LIN {X 0,Y 192.943,Z 262.908,A -85,B 0,C 180,E1 -21964.191,E2 -21964.191} C_VEL
LIN {X 0,Y 193.037,Z 262.919,A -85,B 0,C 180,E1 -21968.387,E2 -21968.387} C_VEL
LIN {X 0,Y 192.808,Z 262.969,A -85,B 0,C 180,E1 -21972.646,E2 -21972.646} C_VEL
LIN {X 0,Y 192.733,Z 262.955,A -85,B 0,C 180,E1 -21976.974,E2 -21976.974} C_VEL
LIN {X 0,Y 192.605,Z 262.981,A -85,B 0,C 180,E1 -21981.414,E2 -21981.414} C_VEL
LIN {X 0,Y 192.66,Z 262.986,A -85,B 0,C 180,E1 -21984.214,E2 -21984.214} C_VEL
LIN {X 0,Y 192.628,Z 262.969,A -85,B 0,C 180,E1 -21988.874,E2 -21988.874} C_VEL
LIN {X 0,Y 192.623,Z 262.992,A -85,B 0,C 180,E1 -21993.195,E2 -21993.195} C_VEL
LIN {X 0,Y 192.571,Z 262.995,A -85,B 0,C 180,E1 -21998.362,E2 -21998.362} C_VEL
LIN {X 0,Y 192.501,Z 262.997,A -85,B 0,C 180,E1 -22003.094,E2 -22003.094} C_VEL
LIN {X 0,Y 192.501,Z 262.997,A -85,B 0,C 180,E1 -22006.917,E2 -22006.917} C_VEL
LIN {X 0,Y 192.636,Z 263.112,A -85,B 0,C 180,E1 -22011.215,E2 -22011.215} C_VEL
LIN {X 0,Y 193.486,Z 266.81,A -85,B 0,C 180,E1 -22013.229,E2 -22013.229} C_VEL
LIN {X 0,Y 195.559,Z 272.184,A -85,B 0,C 180,E1 -22013.906,E2 -22013.906} C_VEL
LIN {X 0,Y 202.679,Z 290.586,A -85,B 0,C 180,E1 -22015.768,E2 -22015.768} C_VEL
LIN {X 0,Y 207.241,Z 304.045,A -85,B 0,C 180,E1 -22016.961,E2 -22016.961} C_VEL
LIN {X 0,Y 208.938,Z 318.725,A -85,B 0,C 180,E1 -22017.817,E2 -22017.817} C_VEL
LIN {X 0,Y 208.478,Z 329.306,A -85,B 0,C 180,E1 -22018.229,E2 -22018.229} C_VEL
LIN {X 0,Y 207.471,Z 335.115,A -85,B 0,C 180,E1 -22018.369,E2 -22018.369} C_VEL
LIN {X 0,Y 201.296,Z 353.95,A -85,B 0,C 180,E1 -22018.502,E2 -22018.502} C_VEL
LIN {X 0,Y 200.376,Z 359.758,A -85,B 0,C 180,E1 -22018.662,E2 -22018.662} C_VEL
LIN {X 0,Y 199.212,Z 377.564,A -85,B 0,C 180,E1 -22019.45,E2 -22019.45} C_VEL
LIN {X 0,Y 198.023,Z 389.93,A -85,B 0,C 180,E1 -22020.35,E2 -22020.35} C_VEL
LIN {X 0,Y 196.332,Z 402.666,A -85,B 0,C 180,E1 -22021.682,E2 -22021.682} C_VEL
LIN {X 0,Y 194.124,Z 414.844,A -85,B 0,C 180,E1 -22023.38,E2 -22023.38} C_VEL
LIN {X 0,Y 192.053,Z 425.896,A -85,B 0,C 180,E1 -22025.398,E2 -22025.398} C_VEL
LIN {X 0,Y 189.821,Z 436.544,A -85,B 0,C 180,E1 -22027.884,E2 -22027.884} C_VEL
LIN {X 0,Y 188.046,Z 444.993,A -85,B 0,C 180,E1 -22030.341,E2 -22030.341} C_VEL
LIN {X 0,Y 186.127,Z 453.853,A -85,B 0,C 180,E1 -22033.545,E2 -22033.545} C_VEL
LIN {X 0,Y 184.71,Z 460.891,A -85,B 0,C 180,E1 -22036.8,E2 -22036.8} C_VEL
LIN {X 0,Y 183.77,Z 466.502,A -85,B 0,C 180,E1 -22040.087,E2 -22040.087} C_VEL
LIN {X 0,Y 183.246,Z 470.863,A -85,B 0,C 180,E1 -22043.389,E2 -22043.389} C_VEL
LIN {X 0,Y 183.046,Z 474.187,A -85,B 0,C 180,E1 -22046.805,E2 -22046.805} C_VEL
LIN {X 0,Y 183.098,Z 476.306,A -85,B 0,C 180,E1 -22049.996,E2 -22049.996} C_VEL
LIN {X 0,Y 182.998,Z 477.475,A -85,B 0,C 180,E1 -22052.916,E2 -22052.916} C_VEL
LIN {X 0,Y 183.265,Z 477.907,A -85,B 0,C 180,E1 -22056.602,E2 -22056.602} C_VEL
LIN {X 0,Y 184.266,Z 476.962,A -85,B 0,C 180,E1 -22060.99,E2 -22060.99} C_VEL
LIN {X 0,Y 186.161,Z 474.469,A -85,B 0,C 180,E1 -22065.319,E2 -22065.319} C_VEL
LIN {X 0,Y 188.203,Z 471.507,A -85,B 0,C 180,E1 -22068.502,E2 -22068.502} C_VEL
LIN {X 0,Y 191.01,Z 467.529,A -85,B 0,C 180,E1 -22071.584,E2 -22071.584} C_VEL
LIN {X 0,Y 194.38,Z 462.447,A -85,B 0,C 180,E1 -22074.565,E2 -22074.565} C_VEL
LIN {X 0,Y 197.93,Z 456.142,A -85,B 0,C 180,E1 -22077.486,E2 -22077.486} C_VEL
LIN {X 0,Y 202.122,Z 448.306,A -85,B 0,C 180,E1 -22080.273,E2 -22080.273} C_VEL
LIN {X 0,Y 206.964,Z 438.674,A -85,B 0,C 180,E1 -22082.906,E2 -22082.906} C_VEL
LIN {X 0,Y 211.367,Z 428.74,A -85,B 0,C 180,E1 -22084.995,E2 -22084.995} C_VEL
LIN {X 0,Y 215.507,Z 417.692,A -85,B 0,C 180,E1 -22086.811,E2 -22086.811} C_VEL
LIN {X 0,Y 219.025,Z 406.97,A -85,B 0,C 180,E1 -22088.143,E2 -22088.143} C_VEL
LIN {X 0,Y 222.085,Z 395.375,A -85,B 0,C 180,E1 -22089.26,E2 -22089.26} C_VEL
LIN {X 0,Y 224.719,Z 382.374,A -85,B 0,C 180,E1 -22090.145,E2 -22090.145} C_VEL
LIN {X 0,Y 226.623,Z 368.194,A -85,B 0,C 180,E1 -22090.777,E2 -22090.777} C_VEL
LIN {X 0,Y 229.852,Z 331.704,A -85,B 0,C 180,E1 -22092.063,E2 -22092.063} C_VEL
LIN {X 0,Y 226.618,Z 323.344,A -85,B 0,C 180,E1 -22093.846,E2 -22093.846} C_VEL
LIN {X 0,Y 222.913,Z 315.251,A -85,B 0,C 180,E1 -22096.011,E2 -22096.011} C_VEL
LIN {X 0,Y 219.308,Z 308.517,A -85,B 0,C 180,E1 -22098.305,E2 -22098.305} C_VEL
LIN {X 0,Y 217.579,Z 305.452,A -85,B 0,C 180,E1 -22099.541,E2 -22099.541} C_VEL
LIN {X 0,Y 215.143,Z 301.303,A -85,B 0,C 180,E1 -22101.43,E2 -22101.43} C_VEL
LIN {X 0,Y 212.377,Z 296.664,A -85,B 0,C 180,E1 -22103.944,E2 -22103.944} C_VEL
LIN {X 0,Y 208.556,Z 290.768,A -85,B 0,C 180,E1 -22108.479,E2 -22108.479} C_VEL
LIN {X 0,Y 205.607,Z 286.729,A -85,B 0,C 180,E1 -22115.057,E2 -22115.057} C_VEL
LIN {X 0,Y 205.277,Z 286.197,A -85,B 0,C 180,E1 -22117.864,E2 -22117.864} C_VEL
LIN {X 0,Y 206.045,Z 286.988,A -85,B 0,C 180,E1 -22122.742,E2 -22122.742} C_VEL
LIN {X 0,Y 209.265,Z 290.496,A -85,B 0,C 180,E1 -22128.554,E2 -22128.554} C_VEL
LIN {X 0,Y 212.901,Z 295.629,A -85,B 0,C 180,E1 -22132.601,E2 -22132.601} C_VEL
LIN {X 0,Y 215.785,Z 299.597,A -85,B 0,C 180,E1 -22135.063,E2 -22135.063} C_VEL
LIN {X 0,Y 218.709,Z 304.458,A -85,B 0,C 180,E1 -22137.267,E2 -22137.267} C_VEL
LIN {X 0,Y 223.96,Z 314.057,A -85,B 0,C 180,E1 -22140.63,E2 -22140.63} C_VEL
LIN {X 0,Y 227.578,Z 321.869,A -85,B 0,C 180,E1 -22142.69,E2 -22142.69} C_VEL
LIN {X 0,Y 230.089,Z 328.091,A -85,B 0,C 180,E1 -22144.05,E2 -22144.05} C_VEL
LIN {X 0,Y 226.135,Z 370.908,A -85,B 0,C 180,E1 -22145.586,E2 -22145.586} C_VEL
LIN {X 0,Y 224.019,Z 383.993,A -85,B 0,C 180,E1 -22146.304,E2 -22146.304} C_VEL
LIN {X 0,Y 221.324,Z 396.216,A -85,B 0,C 180,E1 -22147.285,E2 -22147.285} C_VEL
LIN {X 0,Y 217.858,Z 408.634,A -85,B 0,C 180,E1 -22148.685,E2 -22148.685} C_VEL
LIN {X 0,Y 213.843,Z 420.129,A -85,B 0,C 180,E1 -22150.369,E2 -22150.369} C_VEL
LIN {X 0,Y 210.115,Z 429.29,A -85,B 0,C 180,E1 -22152.088,E2 -22152.088} C_VEL
LIN {X 0,Y 206.133,Z 437.969,A -85,B 0,C 180,E1 -22154.132,E2 -22154.132} C_VEL
LIN {X 0,Y 201.879,Z 446.182,A -85,B 0,C 180,E1 -22156.578,E2 -22156.578} C_VEL
LIN {X 0,Y 197.216,Z 454.354,A -85,B 0,C 180,E1 -22159.727,E2 -22159.727} C_VEL
LIN {X 0,Y 193.229,Z 460.737,A -85,B 0,C 180,E1 -22163,E2 -22163} C_VEL
LIN {X 0,Y 189.936,Z 465.541,A -85,B 0,C 180,E1 -22166.343,E2 -22166.343} C_VEL
LIN {X 0,Y 187.035,Z 469.436,A -85,B 0,C 180,E1 -22170.212,E2 -22170.212} C_VEL
LIN {X 0,Y 185.258,Z 471.55,A -85,B 0,C 180,E1 -22173.434,E2 -22173.434} C_VEL
LIN {X 0,Y 183.606,Z 472.976,A -85,B 0,C 180,E1 -22177.745,E2 -22177.745} C_VEL
LIN {X 0,Y 183,Z 473.017,A -85,B 0,C 180,E1 -22180.736,E2 -22180.736} C_VEL
LIN {X 0,Y 182.634,Z 472.317,A -85,B 0,C 180,E1 -22183.817,E2 -22183.817} C_VEL
LIN {X 0,Y 182.538,Z 470.782,A -85,B 0,C 180,E1 -22186.989,E2 -22186.989} C_VEL
LIN {X 0,Y 182.746,Z 468.284,A -85,B 0,C 180,E1 -22190.251,E2 -22190.251} C_VEL
LIN {X 0,Y 183.32,Z 464.679,A -85,B 0,C 180,E1 -22193.589,E2 -22193.589} C_VEL
LIN {X 0,Y 184.166,Z 459.647,A -85,B 0,C 180,E1 -22197.059,E2 -22197.059} C_VEL
LIN {X 0,Y 185.489,Z 452.98,A -85,B 0,C 180,E1 -22200.591,E2 -22200.591} C_VEL
LIN {X 0,Y 187.055,Z 445.451,A -85,B 0,C 180,E1 -22203.738,E2 -22203.738} C_VEL
LIN {X 0,Y 188.731,Z 437.834,A -85,B 0,C 180,E1 -22206.304,E2 -22206.304} C_VEL
LIN {X 0,Y 190.794,Z 428.078,A -85,B 0,C 180,E1 -22208.956,E2 -22208.956} C_VEL
LIN {X 0,Y 192.965,Z 417.676,A -85,B 0,C 180,E1 -22211.199,E2 -22211.199} C_VEL
LIN {X 0,Y 194.794,Z 407.505,A -85,B 0,C 180,E1 -22212.958,E2 -22212.958} C_VEL
LIN {X 0,Y 196.748,Z 395.175,A -85,B 0,C 180,E1 -22214.614,E2 -22214.614} C_VEL
LIN {X 0,Y 198.396,Z 381.535,A -85,B 0,C 180,E1 -22215.941,E2 -22215.941} C_VEL
LIN {X 0,Y 199.661,Z 367.958,A -85,B 0,C 180,E1 -22216.81,E2 -22216.81} C_VEL
LIN {X 0,Y 202.729,Z 307.987,A -85,B 0,C 180,E1 -22219.215,E2 -22219.215} C_VEL
LIN {X 0,Y 195.715,Z 287.677,A -85,B 0,C 180,E1 -22221.114,E2 -22221.114} C_VEL
LIN {X 0,Y 189.308,Z 271.417,A -85,B 0,C 180,E1 -22222.874,E2 -22222.874} C_VEL
LIN {X 0,Y 186.118,Z 264.918,A -85,B 0,C 180,E1 -22223.771,E2 -22223.771} C_VEL
LIN {X 0,Y 185.888,Z 263.91,A -85,B 0,C 180,E1 -22224.24,E2 -22224.24} C_VEL
LIN {X 0,Y 186.167,Z 263.797,A -85,B 0,C 180,E1 -22227.84,E2 -22227.84} C_VEL
LIN {X 0,Y 186.349,Z 263.764,A -85,B 0,C 180,E1 -22230.004,E2 -22230.004} C_VEL
LIN {X 0,Y 185.876,Z 263.818,A -85,B 0,C 180,E1 -22234.341,E2 -22234.341} C_VEL
LIN {X 0,Y 185.949,Z 263.814,A -85,B 0,C 180,E1 -22238.699,E2 -22238.699} C_VEL
LIN {X 0,Y 185.669,Z 263.855,A -85,B 0,C 180,E1 -22243.131,E2 -22243.131} C_VEL
LIN {X 0,Y 185.633,Z 263.839,A -85,B 0,C 180,E1 -22247.634,E2 -22247.634} C_VEL
LIN {X 0,Y 185.526,Z 263.875,A -85,B 0,C 180,E1 -22252.264,E2 -22252.264} C_VEL
LIN {X 0,Y 185.511,Z 263.851,A -85,B 0,C 180,E1 -22257.044,E2 -22257.044} C_VEL
LIN {X 0,Y 185.533,Z 263.838,A -85,B 0,C 180,E1 -22259.505,E2 -22259.505} C_VEL
LIN {X 0,Y 185.479,Z 263.881,A -85,B 0,C 180,E1 -22264.64,E2 -22264.64} C_VEL
LIN {X 0,Y 185.53,Z 263.87,A -85,B 0,C 180,E1 -22267.327,E2 -22267.327} C_VEL
LIN {X 0,Y 185.526,Z 263.872,A -85,B 0,C 180,E1 -22270.771,E2 -22270.771} C_VEL
LIN {X 0,Y 185.554,Z 263.861,A -85,B 0,C 180,E1 -22276.029,E2 -22276.029} C_VEL
LIN {X 0,Y 185.553,Z 263.869,A -85,B 0,C 180,E1 -22279.939,E2 -22279.939} C_VEL
LIN {X 0,Y 185.551,Z 263.868,A -85,B 0,C 180,E1 -22282.719,E2 -22282.719} C_VEL
LIN {X 0,Y 185.521,Z 263.872,A -85,B 0,C 180,E1 -22287.99,E2 -22287.99} C_VEL
LIN {X 0,Y 185.564,Z 263.87,A -85,B 0,C 180,E1 -22290.592,E2 -22290.592} C_VEL
LIN {X 0,Y 185.568,Z 263.856,A -85,B 0,C 180,E1 -22295.397,E2 -22295.397} C_VEL
LIN {X 0,Y 185.618,Z 263.86,A -85,B 0,C 180,E1 -22301.194,E2 -22301.194} C_VEL
LIN {X 0,Y 185.664,Z 263.844,A -85,B 0,C 180,E1 -22304.65,E2 -22304.65} C_VEL
LIN {X 0,Y 185.889,Z 263.83,A -85,B 0,C 180,E1 -22309.435,E2 -22309.435} C_VEL
LIN {X 0,Y 185.936,Z 263.809,A -85,B 0,C 180,E1 -22313.504,E2 -22313.504} C_VEL
LIN {X 0,Y 186.187,Z 263.794,A -85,B 0,C 180,E1 -22317.851,E2 -22317.851} C_VEL
LIN {X 0,Y 186.388,Z 263.76,A -85,B 0,C 180,E1 -22320.014,E2 -22320.014} C_VEL
LIN {X 0,Y 185.892,Z 263.783,A -85,B 0,C 180,E1 -22324.35,E2 -22324.35} C_VEL
LIN {X 0,Y 185.987,Z 263.798,A -85,B 0,C 180,E1 -22328.707,E2 -22328.707} C_VEL
LIN {X 0,Y 185.734,Z 263.848,A -85,B 0,C 180,E1 -22333.136,E2 -22333.136} C_VEL
LIN {X 0,Y 185.672,Z 263.828,A -85,B 0,C 180,E1 -22337.64,E2 -22337.64} C_VEL
LIN {X 0,Y 185.577,Z 263.863,A -85,B 0,C 180,E1 -22342.268,E2 -22342.268} C_VEL
LIN {X 0,Y 185.603,Z 263.867,A -85,B 0,C 180,E1 -22344.656,E2 -22344.656} C_VEL
LIN {X 0,Y 185.571,Z 263.849,A -85,B 0,C 180,E1 -22349.509,E2 -22349.509} C_VEL
LIN {X 0,Y 185.526,Z 263.867,A -85,B 0,C 180,E1 -22354.641,E2 -22354.641} C_VEL
LIN {X 0,Y 185.53,Z 263.86,A -85,B 0,C 180,E1 -22357.322,E2 -22357.322} C_VEL
LIN {X 0,Y 185.487,Z 263.875,A -85,B 0,C 180,E1 -22360.726,E2 -22360.726} C_VEL
LIN {X 0,Y 185.471,Z 263.874,A -85,B 0,C 180,E1 -22366.068,E2 -22366.068} C_VEL
LIN {X 0,Y 185.54,Z 263.987,A -85,B 0,C 180,E1 -22370.564,E2 -22370.564} C_VEL
LIN {X 0,Y 186.251,Z 266.867,A -85,B 0,C 180,E1 -22372.141,E2 -22372.141} C_VEL
LIN {X 0,Y 194.045,Z 286.32,A -85,B 0,C 180,E1 -22374.371,E2 -22374.371} C_VEL
LIN {X 0,Y 200.783,Z 305.431,A -85,B 0,C 180,E1 -22376.209,E2 -22376.209} C_VEL
LIN {X 0,Y 202.406,Z 318.992,A -85,B 0,C 180,E1 -22377.042,E2 -22377.042} C_VEL
LIN {X 0,Y 200.376,Z 359.758,A -85,B 0,C 180,E1 -22378.662,E2 -22378.662} C_VEL
LIN {X 0,Y 199.401,Z 365.56,A -85,B 0,C 180,E1 -22378.812,E2 -22378.812} C_VEL
LIN {X 0,Y 196.096,Z 374.906,A -85,B 0,C 180,E1 -22378.919,E2 -22378.919} C_VEL
LIN {X 0,Y 192.64,Z 384.148,A -85,B 0,C 180,E1 -22379.212,E2 -22379.212} C_VEL
LIN {X 0,Y 191.389,Z 389.784,A -85,B 0,C 180,E1 -22379.607,E2 -22379.607} C_VEL
LIN {X 0,Y 189.738,Z 401.969,A -85,B 0,C 180,E1 -22380.908,E2 -22380.908} C_VEL
LIN {X 0,Y 187.446,Z 414.254,A -85,B 0,C 180,E1 -22382.655,E2 -22382.655} C_VEL
LIN {X 0,Y 185.304,Z 425.407,A -85,B 0,C 180,E1 -22384.739,E2 -22384.739} C_VEL
LIN {X 0,Y 183.36,Z 434.733,A -85,B 0,C 180,E1 -22386.938,E2 -22386.938} C_VEL
LIN {X 0,Y 181.356,Z 443.789,A -85,B 0,C 180,E1 -22389.584,E2 -22389.584} C_VEL
LIN {X 0,Y 179.309,Z 452.844,A -85,B 0,C 180,E1 -22392.901,E2 -22392.901} C_VEL
LIN {X 0,Y 177.746,Z 460.082,A -85,B 0,C 180,E1 -22396.273,E2 -22396.273} C_VEL
LIN {X 0,Y 176.773,Z 465.831,A -85,B 0,C 180,E1 -22399.69,E2 -22399.69} C_VEL
LIN {X 0,Y 176.174,Z 470.315,A -85,B 0,C 180,E1 -22403.123,E2 -22403.123} C_VEL
LIN {X 0,Y 175.945,Z 474.169,A -85,B 0,C 180,E1 -22407.192,E2 -22407.192} C_VEL
LIN {X 0,Y 176.01,Z 476.003,A -85,B 0,C 180,E1 -22409.996,E2 -22409.996} C_VEL
LIN {X 0,Y 175.927,Z 477.13,A -85,B 0,C 180,E1 -22412.685,E2 -22412.685} C_VEL
LIN {X 0,Y 176.197,Z 477.809,A -85,B 0,C 180,E1 -22416.869,E2 -22416.869} C_VEL
LIN {X 0,Y 176.661,Z 477.609,A -85,B 0,C 180,E1 -22419.152,E2 -22419.152} C_VEL
LIN {X 0,Y 178.159,Z 476.029,A -85,B 0,C 180,E1 -22423.687,E2 -22423.687} C_VEL
LIN {X 0,Y 179.295,Z 474.667,A -85,B 0,C 180,E1 -22425.921,E2 -22425.921} C_VEL
LIN {X 0,Y 181.486,Z 471.823,A -85,B 0,C 180,E1 -22429.213,E2 -22429.213} C_VEL
LIN {X 0,Y 184.449,Z 467.979,A -85,B 0,C 180,E1 -22432.393,E2 -22432.393} C_VEL
LIN {X 0,Y 187.984,Z 463.04,A -85,B 0,C 180,E1 -22435.459,E2 -22435.459} C_VEL
LIN {X 0,Y 191.723,Z 456.951,A -85,B 0,C 180,E1 -22438.455,E2 -22438.455} C_VEL
LIN {X 0,Y 196.098,Z 449.433,A -85,B 0,C 180,E1 -22441.305,E2 -22441.305} C_VEL
LIN {X 0,Y 201.13,Z 440.041,A -85,B 0,C 180,E1 -22443.988,E2 -22443.988} C_VEL
LIN {X 0,Y 206.175,Z 429.387,A -85,B 0,C 180,E1 -22446.314,E2 -22446.314} C_VEL
LIN {X 0,Y 210.502,Z 418.502,A -85,B 0,C 180,E1 -22448.14,E2 -22448.14} C_VEL
LIN {X 0,Y 214.636,Z 406.416,A -85,B 0,C 180,E1 -22449.675,E2 -22449.675} C_VEL
LIN {X 0,Y 217.86,Z 394.75,A -85,B 0,C 180,E1 -22450.782,E2 -22450.782} C_VEL
LIN {X 0,Y 220.676,Z 381.375,A -85,B 0,C 180,E1 -22451.664,E2 -22451.664} C_VEL
LIN {X 0,Y 222.481,Z 368.302,A -85,B 0,C 180,E1 -22452.246,E2 -22452.246} C_VEL
LIN {X 0,Y 225.592,Z 334.403,A -85,B 0,C 180,E1 -22453.456,E2 -22453.456} C_VEL
LIN {X 0,Y 222.567,Z 326.486,A -85,B 0,C 180,E1 -22455.273,E2 -22455.273} C_VEL
LIN {X 0,Y 219.169,Z 319.127,A -85,B 0,C 180,E1 -22457.448,E2 -22457.448} C_VEL
LIN {X 0,Y 215.922,Z 312.59,A -85,B 0,C 180,E1 -22459.792,E2 -22459.792} C_VEL
LIN {X 0,Y 213.028,Z 307.584,A -85,B 0,C 180,E1 -22462.111,E2 -22462.111} C_VEL
LIN {X 0,Y 210.548,Z 303.185,A -85,B 0,C 180,E1 -22464.544,E2 -22464.544} C_VEL
LIN {X 0,Y 207.166,Z 297.618,A -85,B 0,C 180,E1 -22468.823,E2 -22468.823} C_VEL
LIN {X 0,Y 204.482,Z 293.758,A -85,B 0,C 180,E1 -22475.153,E2 -22475.153} C_VEL
LIN {X 0,Y 204.165,Z 293.251,A -85,B 0,C 180,E1 -22478.334,E2 -22478.334} C_VEL
LIN {X 0,Y 204.902,Z 293.994,A -85,B 0,C 180,E1 -22482.643,E2 -22482.643} C_VEL
LIN {X 0,Y 207.812,Z 297.302,A -85,B 0,C 180,E1 -22488.157,E2 -22488.157} C_VEL
LIN {X 0,Y 211.121,Z 302.256,A -85,B 0,C 180,E1 -22492.065,E2 -22492.065} C_VEL
LIN {X 0,Y 214.233,Z 306.793,A -85,B 0,C 180,E1 -22494.856,E2 -22494.856} C_VEL
LIN {X 0,Y 216.427,Z 310.764,A -85,B 0,C 180,E1 -22496.588,E2 -22496.588} C_VEL
LIN {X 0,Y 220.877,Z 319.222,A -85,B 0,C 180,E1 -22499.646,E2 -22499.646} C_VEL
LIN {X 0,Y 224.258,Z 326.949,A -85,B 0,C 180,E1 -22501.754,E2 -22501.754} C_VEL
LIN {X 0,Y 225.869,Z 330.944,A -85,B 0,C 180,E1 -22502.676,E2 -22502.676} C_VEL
LIN {X 0,Y 221.927,Z 371.369,A -85,B 0,C 180,E1 -22504.127,E2 -22504.127} C_VEL
LIN {X 0,Y 219.743,Z 384.284,A -85,B 0,C 180,E1 -22504.849,E2 -22504.849} C_VEL
LIN {X 0,Y 216.995,Z 396.09,A -85,B 0,C 180,E1 -22505.796,E2 -22505.796} C_VEL
LIN {X 0,Y 213.768,Z 407.208,A -85,B 0,C 180,E1 -22507.016,E2 -22507.016} C_VEL
LIN {X 0,Y 209.65,Z 418.687,A -85,B 0,C 180,E1 -22508.663,E2 -22508.663} C_VEL
LIN {X 0,Y 205.282,Z 429.112,A -85,B 0,C 180,E1 -22510.589,E2 -22510.589} C_VEL
LIN {X 0,Y 200.874,Z 438.27,A -85,B 0,C 180,E1 -22512.759,E2 -22512.759} C_VEL
LIN {X 0,Y 196.084,Z 446.97,A -85,B 0,C 180,E1 -22515.419,E2 -22515.419} C_VEL
LIN {X 0,Y 191.199,Z 454.924,A -85,B 0,C 180,E1 -22518.602,E2 -22518.602} C_VEL
LIN {X 0,Y 186.853,Z 461.342,A -85,B 0,C 180,E1 -22522.077,E2 -22522.077} C_VEL
LIN {X 0,Y 182.891,Z 466.644,A -85,B 0,C 180,E1 -22526.051,E2 -22526.051} C_VEL
LIN {X 0,Y 180.551,Z 469.49,A -85,B 0,C 180,E1 -22529.096,E2 -22529.096} C_VEL
LIN {X 0,Y 178.038,Z 472.143,A -85,B 0,C 180,E1 -22533.528,E2 -22533.528} C_VEL
LIN {X 0,Y 176.611,Z 473.118,A -85,B 0,C 180,E1 -22537.27,E2 -22537.27} C_VEL
LIN {X 0,Y 175.909,Z 473.08,A -85,B 0,C 180,E1 -22540.622,E2 -22540.622} C_VEL
LIN {X 0,Y 175.524,Z 472.212,A -85,B 0,C 180,E1 -22543.892,E2 -22543.892} C_VEL
LIN {X 0,Y 175.439,Z 470.584,A -85,B 0,C 180,E1 -22547.083,E2 -22547.083} C_VEL
LIN {X 0,Y 175.652,Z 468.211,A -85,B 0,C 180,E1 -22550.201,E2 -22550.201} C_VEL
LIN {X 0,Y 176.163,Z 465.057,A -85,B 0,C 180,E1 -22553.249,E2 -22553.249} C_VEL
LIN {X 0,Y 177.069,Z 459.663,A -85,B 0,C 180,E1 -22557.151,E2 -22557.151} C_VEL
LIN {X 0,Y 178.535,Z 452.539,A -85,B 0,C 180,E1 -22561.043,E2 -22561.043} C_VEL
LIN {X 0,Y 179.934,Z 445.925,A -85,B 0,C 180,E1 -22563.901,E2 -22563.901} C_VEL
LIN {X 0,Y 181.966,Z 437.067,A -85,B 0,C 180,E1 -22566.984,E2 -22566.984} C_VEL
LIN {X 0,Y 184.045,Z 427.574,A -85,B 0,C 180,E1 -22569.612,E2 -22569.612} C_VEL
LIN {X 0,Y 186.201,Z 417.513,A -85,B 0,C 180,E1 -22571.84,E2 -22571.84} C_VEL
LIN {X 0,Y 188.145,Z 407.091,A -85,B 0,C 180,E1 -22573.689,E2 -22573.689} C_VEL
LIN {X 0,Y 190.017,Z 395.658,A -85,B 0,C 180,E1 -22575.273,E2 -22575.273} C_VEL
LIN {X 0,Y 191.719,Z 382.35,A -85,B 0,C 180,E1 -22576.624,E2 -22576.624} C_VEL
LIN {X 0,Y 193.031,Z 368.868,A -85,B 0,C 180,E1 -22577.544,E2 -22577.544} C_VEL
LIN {X 0,Y 196.268,Z 309.645,A -85,B 0,C 180,E1 -22579.989,E2 -22579.989} C_VEL
LIN {X 0,Y 189.484,Z 290.002,A -85,B 0,C 180,E1 -22581.908,E2 -22581.908} C_VEL
LIN {X 0,Y 183.624,Z 274.948,A -85,B 0,C 180,E1 -22583.59,E2 -22583.59} C_VEL
LIN {X 0,Y 179.128,Z 265.97,A -85,B 0,C 180,E1 -22584.868,E2 -22584.868} C_VEL
LIN {X 0,Y 178.868,Z 264.809,A -85,B 0,C 180,E1 -22585.355,E2 -22585.355} C_VEL
LIN {X 0,Y 179.313,Z 264.64,A -85,B 0,C 180,E1 -22590.004,E2 -22590.004} C_VEL
LIN {X 0,Y 178.823,Z 264.696,A -85,B 0,C 180,E1 -22594.512,E2 -22594.512} C_VEL
LIN {X 0,Y 178.879,Z 264.69,A -85,B 0,C 180,E1 -22599.046,E2 -22599.046} C_VEL
LIN {X 0,Y 178.598,Z 264.739,A -85,B 0,C 180,E1 -22603.661,E2 -22603.661} C_VEL
LIN {X 0,Y 178.569,Z 264.719,A -85,B 0,C 180,E1 -22609.222,E2 -22609.222} C_VEL
LIN {X 0,Y 178.472,Z 264.747,A -85,B 0,C 180,E1 -22615.125,E2 -22615.125} C_VEL
LIN {X 0,Y 178.477,Z 264.718,A -85,B 0,C 180,E1 -22620.005,E2 -22620.005} C_VEL
LIN {X 0,Y 178.443,Z 264.757,A -85,B 0,C 180,E1 -22624.231,E2 -22624.231} C_VEL
LIN {X 0,Y 178.436,Z 264.747,A -85,B 0,C 180,E1 -22629.068,E2 -22629.068} C_VEL
LIN {X 0,Y 178.468,Z 264.753,A -85,B 0,C 180,E1 -22632.029,E2 -22632.029} C_VEL
LIN {X 0,Y 178.496,Z 264.743,A -85,B 0,C 180,E1 -22635.136,E2 -22635.136} C_VEL
LIN {X 0,Y 178.493,Z 264.743,A -85,B 0,C 180,E1 -22638.432,E2 -22638.432} C_VEL
LIN {X 0,Y 178.465,Z 264.746,A -85,B 0,C 180,E1 -22643.814,E2 -22643.814} C_VEL
LIN {X 0,Y 178.469,Z 264.742,A -85,B 0,C 180,E1 -22646.563,E2 -22646.563} C_VEL
LIN {X 0,Y 178.504,Z 264.748,A -85,B 0,C 180,E1 -22650.024,E2 -22650.024} C_VEL
LIN {X 0,Y 178.507,Z 264.733,A -85,B 0,C 180,E1 -22654.902,E2 -22654.902} C_VEL
LIN {X 0,Y 178.601,Z 264.73,A -85,B 0,C 180,E1 -22661.668,E2 -22661.668} C_VEL
LIN {X 0,Y 178.642,Z 264.728,A -85,B 0,C 180,E1 -22666.363,E2 -22666.363} C_VEL
LIN {X 0,Y 178.906,Z 264.694,A -85,B 0,C 180,E1 -22670.975,E2 -22670.975} C_VEL
LIN {X 0,Y 179.134,Z 264.672,A -85,B 0,C 180,E1 -22677.766,E2 -22677.766} C_VEL
LIN {X 0,Y 179.353,Z 264.635,A -85,B 0,C 180,E1 -22680.015,E2 -22680.015} C_VEL
LIN {X 0,Y 178.841,Z 264.658,A -85,B 0,C 180,E1 -22684.522,E2 -22684.522} C_VEL
LIN {X 0,Y 178.919,Z 264.681,A -85,B 0,C 180,E1 -22689.054,E2 -22689.054} C_VEL
LIN {X 0,Y 178.66,Z 264.729,A -85,B 0,C 180,E1 -22693.666,E2 -22693.666} C_VEL
LIN {X 0,Y 178.576,Z 264.707,A -85,B 0,C 180,E1 -22699.163,E2 -22699.163} C_VEL
LIN {X 0,Y 178.542,Z 264.743,A -85,B 0,C 180,E1 -22705.121,E2 -22705.121} C_VEL
LIN {X 0,Y 178.488,Z 264.741,A -85,B 0,C 180,E1 -22710.804,E2 -22710.804} C_VEL
LIN {X 0,Y 178.512,Z 264.745,A -85,B 0,C 180,E1 -22714.226,E2 -22714.226} C_VEL
LIN {X 0,Y 178.416,Z 264.76,A -85,B 0,C 180,E1 -22719.085,E2 -22719.085} C_VEL
LIN {X 0,Y 178.417,Z 264.748,A -85,B 0,C 180,E1 -22722.056,E2 -22722.056} C_VEL
LIN {X 0,Y 178.413,Z 264.76,A -85,B 0,C 180,E1 -22725.175,E2 -22725.175} C_VEL
LIN {X 0,Y 178.457,Z 264.872,A -85,B 0,C 180,E1 -22729.849,E2 -22729.849} C_VEL
LIN {X 0,Y 179.019,Z 266.974,A -85,B 0,C 180,E1 -22730.962,E2 -22730.962} C_VEL
LIN {X 0,Y 186.354,Z 284.848,A -85,B 0,C 180,E1 -22733.148,E2 -22733.148} C_VEL
LIN {X 0,Y 194.013,Z 306.113,A -85,B 0,C 180,E1 -22735.326,E2 -22735.326} C_VEL
LIN {X 0,Y 194.976,Z 311.156,A -85,B 0,C 180,E1 -22735.702,E2 -22735.702} C_VEL
LIN {X 0,Y 195.892,Z 320.242,A -85,B 0,C 180,E1 -22736.26,E2 -22736.26} C_VEL
LIN {X 0,Y 192.915,Z 374.146,A -85,B 0,C 180,E1 -22738.493,E2 -22738.493} C_VEL
LIN {X 0,Y 191.603,Z 388.241,A -85,B 0,C 180,E1 -22739.48,E2 -22739.48} C_VEL
LIN {X 0,Y 191.389,Z 389.784,A -85,B 0,C 180,E1 -22739.607,E2 -22739.607} C_VEL
LIN {X 0,Y 189.977,Z 395.345,A -85,B 0,C 180,E1 -22740.053,E2 -22740.053} C_VEL
LIN {X 0,Y 185.871,Z 404.083,A -85,B 0,C 180,E1 -22740.784,E2 -22740.784} C_VEL
LIN {X 0,Y 181.662,Z 412.499,A -85,B 0,C 180,E1 -22741.769,E2 -22741.769} C_VEL
LIN {X 0,Y 180.106,Z 417.551,A -85,B 0,C 180,E1 -22742.607,E2 -22742.607} C_VEL
LIN {X 0,Y 177.823,Z 428.609,A -85,B 0,C 180,E1 -22744.917,E2 -22744.917} C_VEL
LIN {X 0,Y 175.587,Z 437.995,A -85,B 0,C 180,E1 -22747.37,E2 -22747.37} C_VEL
LIN {X 0,Y 173.806,Z 445.797,A -85,B 0,C 180,E1 -22749.893,E2 -22749.893} C_VEL
LIN {X 0,Y 172.161,Z 453.13,A -85,B 0,C 180,E1 -22752.781,E2 -22752.781} C_VEL
LIN {X 0,Y 170.61,Z 460.275,A -85,B 0,C 180,E1 -22756.295,E2 -22756.295} C_VEL
LIN {X 0,Y 169.493,Z 466.788,A -85,B 0,C 180,E1 -22760.449,E2 -22760.449} C_VEL
LIN {X 0,Y 169,Z 471.027,A -85,B 0,C 180,E1 -22764.028,E2 -22764.028} C_VEL
LIN {X 0,Y 168.853,Z 474.15,A -85,B 0,C 180,E1 -22767.611,E2 -22767.611} C_VEL
LIN {X 0,Y 168.913,Z 475.687,A -85,B 0,C 180,E1 -22769.996,E2 -22769.996} C_VEL
LIN {X 0,Y 168.852,Z 476.749,A -85,B 0,C 180,E1 -22772.381,E2 -22772.381} C_VEL
LIN {X 0,Y 169.153,Z 477.677,A -85,B 0,C 180,E1 -22777.156,E2 -22777.156} C_VEL
LIN {X 0,Y 169.652,Z 477.572,A -85,B 0,C 180,E1 -22779.534,E2 -22779.534} C_VEL
LIN {X 0,Y 170.324,Z 477.064,A -85,B 0,C 180,E1 -22781.902,E2 -22781.902} C_VEL
LIN {X 0,Y 172.45,Z 474.852,A -85,B 0,C 180,E1 -22786.571,E2 -22786.571} C_VEL
LIN {X 0,Y 174.807,Z 472.138,A -85,B 0,C 180,E1 -22789.978,E2 -22789.978} C_VEL
LIN {X 0,Y 177.93,Z 468.454,A -85,B 0,C 180,E1 -22793.261,E2 -22793.261} C_VEL
LIN {X 0,Y 181.638,Z 463.703,A -85,B 0,C 180,E1 -22796.416,E2 -22796.416} C_VEL
LIN {X 0,Y 185.574,Z 457.79,A -85,B 0,C 180,E1 -22799.489,E2 -22799.489} C_VEL
LIN {X 0,Y 190.134,Z 450.471,A -85,B 0,C 180,E1 -22802.405,E2 -22802.405} C_VEL
LIN {X 0,Y 195.395,Z 441.423,A -85,B 0,C 180,E1 -22805.129,E2 -22805.129} C_VEL
LIN {X 0,Y 200.647,Z 431.129,A -85,B 0,C 180,E1 -22807.483,E2 -22807.483} C_VEL
LIN {X 0,Y 205.136,Z 420.813,A -85,B 0,C 180,E1 -22809.327,E2 -22809.327} C_VEL
LIN {X 0,Y 209.425,Z 409.348,A -85,B 0,C 180,E1 -22810.868,E2 -22810.868} C_VEL
LIN {X 0,Y 212.985,Z 397.454,A -85,B 0,C 180,E1 -22812.082,E2 -22812.082} C_VEL
LIN {X 0,Y 216.169,Z 383.924,A -85,B 0,C 180,E1 -22813.053,E2 -22813.053} C_VEL
LIN {X 0,Y 218.3,Z 370.001,A -85,B 0,C 180,E1 -22813.714,E2 -22813.714} C_VEL
LIN {X 0,Y 221.476,Z 337.116,A -85,B 0,C 180,E1 -22814.912,E2 -22814.912} C_VEL
LIN {X 0,Y 218.372,Z 328.965,A -85,B 0,C 180,E1 -22816.997,E2 -22816.997} C_VEL
LIN {X 0,Y 214.954,Z 321.517,A -85,B 0,C 180,E1 -22819.468,E2 -22819.468} C_VEL
LIN {X 0,Y 212.475,Z 316.666,A -85,B 0,C 180,E1 -22821.473,E2 -22821.473} C_VEL
LIN {X 0,Y 210.818,Z 313.593,A -85,B 0,C 180,E1 -22822.986,E2 -22822.986} C_VEL
LIN {X 0,Y 208.677,Z 309.609,A -85,B 0,C 180,E1 -22825.225,E2 -22825.225} C_VEL
LIN {X 0,Y 205.643,Z 304.317,A -85,B 0,C 180,E1 -22829.379,E2 -22829.379} C_VEL
LIN {X 0,Y 203.317,Z 300.675,A -85,B 0,C 180,E1 -22835.481,E2 -22835.481} C_VEL
LIN {X 0,Y 203.111,Z 300.31,A -85,B 0,C 180,E1 -22839.095,E2 -22839.095} C_VEL
LIN {X 0,Y 203.828,Z 301.093,A -85,B 0,C 180,E1 -22842.77,E2 -22842.77} C_VEL
LIN {X 0,Y 206.463,Z 304.248,A -85,B 0,C 180,E1 -22847.891,E2 -22847.891} C_VEL
LIN {X 0,Y 209.336,Z 308.846,A -85,B 0,C 180,E1 -22851.498,E2 -22851.498} C_VEL
LIN {X 0,Y 212.325,Z 313.458,A -85,B 0,C 180,E1 -22854.354,E2 -22854.354} C_VEL
LIN {X 0,Y 214.157,Z 316.953,A -85,B 0,C 180,E1 -22855.875,E2 -22855.875} C_VEL
LIN {X 0,Y 218.631,Z 325.956,A -85,B 0,C 180,E1 -22859.146,E2 -22859.146} C_VEL
LIN {X 0,Y 221.758,Z 333.887,A -85,B 0,C 180,E1 -22861.228,E2 -22861.228} C_VEL
LIN {X 0,Y 217.835,Z 372.108,A -85,B 0,C 180,E1 -22862.628,E2 -22862.628} C_VEL
LIN {X 0,Y 215.486,Z 385.259,A -85,B 0,C 180,E1 -22863.376,E2 -22863.376} C_VEL
LIN {X 0,Y 212.748,Z 396.435,A -85,B 0,C 180,E1 -22864.281,E2 -22864.281} C_VEL
LIN {X 0,Y 209.032,Z 408.477,A -85,B 0,C 180,E1 -22865.622,E2 -22865.622} C_VEL
LIN {X 0,Y 204.604,Z 420.102,A -85,B 0,C 180,E1 -22867.332,E2 -22867.332} C_VEL
LIN {X 0,Y 199.982,Z 430.381,A -85,B 0,C 180,E1 -22869.306,E2 -22869.306} C_VEL
LIN {X 0,Y 195.035,Z 439.837,A -85,B 0,C 180,E1 -22871.668,E2 -22871.668} C_VEL
LIN {X 0,Y 190.081,Z 448.223,A -85,B 0,C 180,E1 -22874.352,E2 -22874.352} C_VEL
LIN {X 0,Y 184.86,Z 456.096,A -85,B 0,C 180,E1 -22877.69,E2 -22877.69} C_VEL
LIN {X 0,Y 180.651,Z 461.859,A -85,B 0,C 180,E1 -22880.995,E2 -22880.995} C_VEL
LIN {X 0,Y 177.221,Z 466.082,A -85,B 0,C 180,E1 -22884.213,E2 -22884.213} C_VEL
LIN {X 0,Y 174.392,Z 469.284,A -85,B 0,C 180,E1 -22887.561,E2 -22887.561} C_VEL
LIN {X 0,Y 171.516,Z 472.084,A -85,B 0,C 180,E1 -22892.166,E2 -22892.166} C_VEL
LIN {X 0,Y 170.136,Z 473.031,A -85,B 0,C 180,E1 -22895.31,E2 -22895.31} C_VEL
LIN {X 0,Y 169.183,Z 473.301,A -85,B 0,C 180,E1 -22898.521,E2 -22898.521} C_VEL
LIN {X 0,Y 168.632,Z 472.82,A -85,B 0,C 180,E1 -22901.798,E2 -22901.798} C_VEL
LIN {X 0,Y 168.361,Z 471.528,A -85,B 0,C 180,E1 -22905.179,E2 -22905.179} C_VEL
LIN {X 0,Y 168.39,Z 469.335,A -85,B 0,C 180,E1 -22908.671,E2 -22908.671} C_VEL
LIN {X 0,Y 168.867,Z 466.124,A -85,B 0,C 180,E1 -22912.225,E2 -22912.225} C_VEL
LIN {X 0,Y 169.625,Z 461.604,A -85,B 0,C 180,E1 -22915.926,E2 -22915.926} C_VEL
LIN {X 0,Y 170.807,Z 455.518,A -85,B 0,C 180,E1 -22919.738,E2 -22919.738} C_VEL
LIN {X 0,Y 172.47,Z 448.036,A -85,B 0,C 180,E1 -22923.374,E2 -22923.374} C_VEL
LIN {X 0,Y 174.617,Z 438.737,A -85,B 0,C 180,E1 -22926.895,E2 -22926.895} C_VEL
LIN {X 0,Y 176.928,Z 428.746,A -85,B 0,C 180,E1 -22929.865,E2 -22929.865} C_VEL
LIN {X 0,Y 179.225,Z 418.262,A -85,B 0,C 180,E1 -22932.312,E2 -22932.312} C_VEL
LIN {X 0,Y 181.501,Z 406.649,A -85,B 0,C 180,E1 -22934.446,E2 -22934.446} C_VEL
LIN {X 0,Y 183.536,Z 394.349,A -85,B 0,C 180,E1 -22936.157,E2 -22936.157} C_VEL
LIN {X 0,Y 185.269,Z 380.688,A -85,B 0,C 180,E1 -22937.543,E2 -22937.543} C_VEL
LIN {X 0,Y 186.578,Z 367.092,A -85,B 0,C 180,E1 -22938.427,E2 -22938.427} C_VEL
LIN {X 0,Y 189.704,Z 310.877,A -85,B 0,C 180,E1 -22940.826,E2 -22940.826} C_VEL
LIN {X 0,Y 183.352,Z 292.548,A -85,B 0,C 180,E1 -22942.709,E2 -22942.709} C_VEL
LIN {X 0,Y 177.935,Z 278.507,A -85,B 0,C 180,E1 -22944.338,E2 -22944.338} C_VEL
LIN {X 0,Y 172.131,Z 266.958,A -85,B 0,C 180,E1 -22946.053,E2 -22946.053} C_VEL
LIN {X 0,Y 171.895,Z 265.696,A -85,B 0,C 180,E1 -22946.561,E2 -22946.561} C_VEL
LIN {X 0,Y 172.276,Z 265.516,A -85,B 0,C 180,E1 -22950.004,E2 -22950.004} C_VEL
LIN {X 0,Y 171.771,Z 265.575,A -85,B 0,C 180,E1 -22954.698,E2 -22954.698} C_VEL
LIN {X 0,Y 171.815,Z 265.566,A -85,B 0,C 180,E1 -22959.421,E2 -22959.421} C_VEL
LIN {X 0,Y 171.515,Z 265.62,A -85,B 0,C 180,E1 -22964.236,E2 -22964.236} C_VEL
LIN {X 0,Y 171.488,Z 265.602,A -85,B 0,C 180,E1 -22969.565,E2 -22969.565} C_VEL
LIN {X 0,Y 171.411,Z 265.621,A -85,B 0,C 180,E1 -22975.619,E2 -22975.619} C_VEL
LIN {X 0,Y 171.395,Z 265.604,A -85,B 0,C 180,E1 -22980.597,E2 -22980.597} C_VEL
LIN {X 0,Y 171.363,Z 265.639,A -85,B 0,C 180,E1 -22985.046,E2 -22985.046} C_VEL
LIN {X 0,Y 171.39,Z 265.624,A -85,B 0,C 180,E1 -22988.85,E2 -22988.85} C_VEL
LIN {X 0,Y 171.417,Z 265.63,A -85,B 0,C 180,E1 -22994.191,E2 -22994.191} C_VEL
LIN {X 0,Y 171.411,Z 265.629,A -85,B 0,C 180,E1 -22999.027,E2 -22999.027} C_VEL
LIN {X 0,Y 171.422,Z 265.63,A -85,B 0,C 180,E1 -23002.073,E2 -23002.073} C_VEL
LIN {X 0,Y 171.398,Z 265.631,A -85,B 0,C 180,E1 -23007.809,E2 -23007.809} C_VEL
LIN {X 0,Y 171.431,Z 265.63,A -85,B 0,C 180,E1 -23010.551,E2 -23010.551} C_VEL
LIN {X 0,Y 171.429,Z 265.619,A -85,B 0,C 180,E1 -23015.816,E2 -23015.816} C_VEL
LIN {X 0,Y 171.501,Z 265.62,A -85,B 0,C 180,E1 -23020.88,E2 -23020.88} C_VEL
LIN {X 0,Y 171.555,Z 265.605,A -85,B 0,C 180,E1 -23025.788,E2 -23025.788} C_VEL
LIN {X 0,Y 171.844,Z 265.573,A -85,B 0,C 180,E1 -23030.601,E2 -23030.601} C_VEL
LIN {X 0,Y 171.794,Z 265.58,A -85,B 0,C 180,E1 -23035.323,E2 -23035.323} C_VEL
LIN {X 0,Y 172.318,Z 265.511,A -85,B 0,C 180,E1 -23040.015,E2 -23040.015} C_VEL
LIN {X 0,Y 171.79,Z 265.533,A -85,B 0,C 180,E1 -23044.708,E2 -23044.708} C_VEL
LIN {X 0,Y 171.858,Z 265.564,A -85,B 0,C 180,E1 -23049.43,E2 -23049.43} C_VEL
LIN {X 0,Y 171.575,Z 265.609,A -85,B 0,C 180,E1 -23054.242,E2 -23054.242} C_VEL
LIN {X 0,Y 171.502,Z 265.588,A -85,B 0,C 180,E1 -23059.511,E2 -23059.511} C_VEL
LIN {X 0,Y 171.469,Z 265.622,A -85,B 0,C 180,E1 -23065.608,E2 -23065.608} C_VEL
LIN {X 0,Y 171.445,Z 265.615,A -85,B 0,C 180,E1 -23070.582,E2 -23070.582} C_VEL
LIN {X 0,Y 171.422,Z 265.618,A -85,B 0,C 180,E1 -23075.044,E2 -23075.044} C_VEL
LIN {X 0,Y 171.372,Z 265.637,A -85,B 0,C 180,E1 -23078.808,E2 -23078.808} C_VEL
LIN {X 0,Y 171.342,Z 265.641,A -85,B 0,C 180,E1 -23084.228,E2 -23084.228} C_VEL
LIN {X 0,Y 171.438,Z 265.883,A -85,B 0,C 180,E1 -23089.175,E2 -23089.175} C_VEL
LIN {X 0,Y 171.769,Z 267.151,A -85,B 0,C 180,E1 -23089.658,E2 -23089.658} C_VEL
LIN {X 0,Y 177.938,Z 281.462,A -85,B 0,C 180,E1 -23091.611,E2 -23091.611} C_VEL
LIN {X 0,Y 185.475,Z 301.584,A -85,B 0,C 180,E1 -23093.878,E2 -23093.878} C_VEL
LIN {X 0,Y 188.3,Z 310.591,A -85,B 0,C 180,E1 -23094.75,E2 -23094.75} C_VEL
LIN {X 0,Y 189.402,Z 321.073,A -85,B 0,C 180,E1 -23095.428,E2 -23095.428} C_VEL
LIN {X 0,Y 186.361,Z 373.625,A -85,B 0,C 180,E1 -23097.673,E2 -23097.673} C_VEL
LIN {X 0,Y 185.13,Z 386.925,A -85,B 0,C 180,E1 -23098.61,E2 -23098.61} C_VEL
LIN {X 0,Y 183.532,Z 398.847,A -85,B 0,C 180,E1 -23099.824,E2 -23099.824} C_VEL
LIN {X 0,Y 181.505,Z 410.249,A -85,B 0,C 180,E1 -23101.365,E2 -23101.365} C_VEL
LIN {X 0,Y 180.106,Z 417.551,A -85,B 0,C 180,E1 -23102.607,E2 -23102.607} C_VEL
LIN {X 0,Y 178.535,Z 422.527,A -85,B 0,C 180,E1 -23103.521,E2 -23103.521} C_VEL
LIN {X 0,Y 174.157,Z 430.135,A -85,B 0,C 180,E1 -23105.006,E2 -23105.006} C_VEL
LIN {X 0,Y 169.657,Z 437.3,A -85,B 0,C 180,E1 -23106.739,E2 -23106.739} C_VEL
LIN {X 0,Y 167.935,Z 441.504,A -85,B 0,C 180,E1 -23108.021,E2 -23108.021} C_VEL
LIN {X 0,Y 166.045,Z 449.213,A -85,B 0,C 180,E1 -23110.847,E2 -23110.847} C_VEL
LIN {X 0,Y 164.118,Z 457.124,A -85,B 0,C 180,E1 -23114.472,E2 -23114.472} C_VEL
LIN {X 0,Y 163.107,Z 462.522,A -85,B 0,C 180,E1 -23117.554,E2 -23117.554} C_VEL
LIN {X 0,Y 162.235,Z 467.7,A -85,B 0,C 180,E1 -23121.275,E2 -23121.275} C_VEL
LIN {X 0,Y 161.832,Z 471.68,A -85,B 0,C 180,E1 -23125.013,E2 -23125.013} C_VEL
LIN {X 0,Y 161.771,Z 474.112,A -85,B 0,C 180,E1 -23128.067,E2 -23128.067} C_VEL
LIN {X 0,Y 161.836,Z 475.307,A -85,B 0,C 180,E1 -23129.996,E2 -23129.996} C_VEL
LIN {X 0,Y 161.771,Z 476.477,A -85,B 0,C 180,E1 -23132.486,E2 -23132.486} C_VEL
LIN {X 0,Y 161.824,Z 477.207,A -85,B 0,C 180,E1 -23134.979,E2 -23134.979} C_VEL
LIN {X 0,Y 162.636,Z 477.503,A -85,B 0,C 180,E1 -23139.949,E2 -23139.949} C_VEL
LIN {X 0,Y 164.366,Z 476.271,A -85,B 0,C 180,E1 -23144.861,E2 -23144.861} C_VEL
LIN {X 0,Y 167.201,Z 473.44,A -85,B 0,C 180,E1 -23149.645,E2 -23149.645} C_VEL
LIN {X 0,Y 170.298,Z 470.232,A -85,B 0,C 180,E1 -23153.078,E2 -23153.078} C_VEL
LIN {X 0,Y 173.981,Z 466.003,A -85,B 0,C 180,E1 -23156.377,E2 -23156.377} C_VEL
LIN {X 0,Y 178.647,Z 459.764,A -85,B 0,C 180,E1 -23160.04,E2 -23160.04} C_VEL
LIN {X 0,Y 183.422,Z 452.875,A -85,B 0,C 180,E1 -23163.088,E2 -23163.088} C_VEL
LIN {X 0,Y 188.81,Z 444.417,A -85,B 0,C 180,E1 -23165.887,E2 -23165.887} C_VEL
LIN {X 0,Y 193.687,Z 435.825,A -85,B 0,C 180,E1 -23168.081,E2 -23168.081} C_VEL
LIN {X 0,Y 198.768,Z 425.395,A -85,B 0,C 180,E1 -23170.181,E2 -23170.181} C_VEL
LIN {X 0,Y 203.12,Z 415.103,A -85,B 0,C 180,E1 -23171.758,E2 -23171.758} C_VEL
LIN {X 0,Y 207.599,Z 402.099,A -85,B 0,C 180,E1 -23173.273,E2 -23173.273} C_VEL
LIN {X 0,Y 210.914,Z 390.325,A -85,B 0,C 180,E1 -23174.235,E2 -23174.235} C_VEL
LIN {X 0,Y 213.555,Z 377.311,A -85,B 0,C 180,E1 -23175.003,E2 -23175.003} C_VEL
LIN {X 0,Y 215.688,Z 359.271,A -85,B 0,C 180,E1 -23175.718,E2 -23175.718} C_VEL
LIN {X 0,Y 217.683,Z 340.238,A -85,B 0,C 180,E1 -23176.372,E2 -23176.372} C_VEL
LIN {X 0,Y 214.654,Z 332.309,A -85,B 0,C 180,E1 -23178.588,E2 -23178.588} C_VEL
LIN {X 0,Y 211.812,Z 325.869,A -85,B 0,C 180,E1 -23180.906,E2 -23180.906} C_VEL
LIN {X 0,Y 209.017,Z 320.202,A -85,B 0,C 180,E1 -23183.52,E2 -23183.52} C_VEL
LIN {X 0,Y 206.856,Z 316.008,A -85,B 0,C 180,E1 -23185.906,E2 -23185.906} C_VEL
LIN {X 0,Y 204.127,Z 310.957,A -85,B 0,C 180,E1 -23189.98,E2 -23189.98} C_VEL
LIN {X 0,Y 202.175,Z 307.651,A -85,B 0,C 180,E1 -23195.674,E2 -23195.674} C_VEL
LIN {X 0,Y 201.986,Z 307.267,A -85,B 0,C 180,E1 -23197.484,E2 -23197.484} C_VEL
LIN {X 0,Y 202.434,Z 307.755,A -85,B 0,C 180,E1 -23201.78,E2 -23201.78} C_VEL
LIN {X 0,Y 205.041,Z 311.068,A -85,B 0,C 180,E1 -23207.506,E2 -23207.506} C_VEL
LIN {X 0,Y 207.672,Z 315.588,A -85,B 0,C 180,E1 -23211.032,E2 -23211.032} C_VEL
LIN {X 0,Y 210.292,Z 319.773,A -85,B 0,C 180,E1 -23213.657,E2 -23213.657} C_VEL
LIN {X 0,Y 211.95,Z 323.218,A -85,B 0,C 180,E1 -23215.173,E2 -23215.173} C_VEL
LIN {X 0,Y 215.935,Z 331.809,A -85,B 0,C 180,E1 -23218.325,E2 -23218.325} C_VEL
LIN {X 0,Y 217.856,Z 336.837,A -85,B 0,C 180,E1 -23219.696,E2 -23219.696} C_VEL
LIN {X 0,Y 214.173,Z 371.835,A -85,B 0,C 180,E1 -23221.013,E2 -23221.013} C_VEL
LIN {X 0,Y 211.842,Z 384.418,A -85,B 0,C 180,E1 -23221.706,E2 -23221.706} C_VEL
LIN {X 0,Y 208.521,Z 397.391,A -85,B 0,C 180,E1 -23222.751,E2 -23222.751} C_VEL
LIN {X 0,Y 204.346,Z 410.008,A -85,B 0,C 180,E1 -23224.201,E2 -23224.201} C_VEL
LIN {X 0,Y 200.045,Z 420.656,A -85,B 0,C 180,E1 -23225.791,E2 -23225.791} C_VEL
LIN {X 0,Y 195.093,Z 431.071,A -85,B 0,C 180,E1 -23227.822,E2 -23227.822} C_VEL
LIN {X 0,Y 189.81,Z 440.617,A -85,B 0,C 180,E1 -23230.252,E2 -23230.252} C_VEL
LIN {X 0,Y 184.911,Z 448.423,A -85,B 0,C 180,E1 -23232.818,E2 -23232.818} C_VEL
LIN {X 0,Y 179.848,Z 455.579,A -85,B 0,C 180,E1 -23235.859,E2 -23235.859} C_VEL
LIN {X 0,Y 174.54,Z 462.332,A -85,B 0,C 180,E1 -23239.795,E2 -23239.795} C_VEL
LIN {X 0,Y 171.121,Z 466.253,A -85,B 0,C 180,E1 -23242.904,E2 -23242.904} C_VEL
LIN {X 0,Y 167.147,Z 470.307,A -85,B 0,C 180,E1 -23247.53,E2 -23247.53} C_VEL
LIN {X 0,Y 164.702,Z 472.338,A -85,B 0,C 180,E1 -23251.424,E2 -23251.424} C_VEL
LIN {X 0,Y 163.082,Z 473.263,A -85,B 0,C 180,E1 -23255.043,E2 -23255.043} C_VEL
LIN {X 0,Y 162.042,Z 473.331,A -85,B 0,C 180,E1 -23258.685,E2 -23258.685} C_VEL
LIN {X 0,Y 161.462,Z 472.58,A -85,B 0,C 180,E1 -23262.279,E2 -23262.279} C_VEL
LIN {X 0,Y 161.246,Z 471.058,A -85,B 0,C 180,E1 -23265.79,E2 -23265.79} C_VEL
LIN {X 0,Y 161.333,Z 468.774,A -85,B 0,C 180,E1 -23269.206,E2 -23269.206} C_VEL
LIN {X 0,Y 161.815,Z 465.685,A -85,B 0,C 180,E1 -23272.557,E2 -23272.557} C_VEL
LIN {X 0,Y 162.693,Z 460.79,A -85,B 0,C 180,E1 -23276.586,E2 -23276.586} C_VEL
LIN {X 0,Y 164.007,Z 454.305,A -85,B 0,C 180,E1 -23280.624,E2 -23280.624} C_VEL
LIN {X 0,Y 165.648,Z 447.11,A -85,B 0,C 180,E1 -23284.125,E2 -23284.125} C_VEL
LIN {X 0,Y 167.587,Z 439.07,A -85,B 0,C 180,E1 -23287.259,E2 -23287.259} C_VEL
LIN {X 0,Y 170.007,Z 429.018,A -85,B 0,C 180,E1 -23290.378,E2 -23290.378} C_VEL
LIN {X 0,Y 172.594,Z 417.534,A -85,B 0,C 180,E1 -23293.139,E2 -23293.139} C_VEL
LIN {X 0,Y 174.804,Z 406.548,A -85,B 0,C 180,E1 -23295.204,E2 -23295.204} C_VEL
LIN {X 0,Y 176.887,Z 394.387,A -85,B 0,C 180,E1 -23296.944,E2 -23296.944} C_VEL
LIN {X 0,Y 178.685,Z 380.698,A -85,B 0,C 180,E1 -23298.375,E2 -23298.375} C_VEL
LIN {X 0,Y 180.026,Z 367.264,A -85,B 0,C 180,E1 -23299.274,E2 -23299.274} C_VEL
LIN {X 0,Y 183.287,Z 312.629,A -85,B 0,C 180,E1 -23301.667,E2 -23301.667} C_VEL
LIN {X 0,Y 176.297,Z 292.269,A -85,B 0,C 180,E1 -23303.868,E2 -23303.868} C_VEL
LIN {X 0,Y 171.889,Z 281.15,A -85,B 0,C 180,E1 -23305.259,E2 -23305.259} C_VEL
LIN {X 0,Y 165.179,Z 267.509,A -85,B 0,C 180,E1 -23307.413,E2 -23307.413} C_VEL
LIN {X 0,Y 165.055,Z 266.497,A -85,B 0,C 180,E1 -23307.945,E2 -23307.945} C_VEL
LIN {X 0,Y 165.239,Z 266.392,A -85,B 0,C 180,E1 -23310.004,E2 -23310.004} C_VEL
LIN {X 0,Y 164.719,Z 266.453,A -85,B 0,C 180,E1 -23314.899,E2 -23314.899} C_VEL
LIN {X 0,Y 164.787,Z 266.459,A -85,B 0,C 180,E1 -23317.355,E2 -23317.355} C_VEL
LIN {X 0,Y 164.685,Z 266.452,A -85,B 0,C 180,E1 -23321.132,E2 -23321.132} C_VEL
LIN {X 0,Y 164.424,Z 266.478,A -85,B 0,C 180,E1 -23327.414,E2 -23327.414} C_VEL
LIN {X 0,Y 164.423,Z 266.484,A -85,B 0,C 180,E1 -23330,E2 -23330} C_VEL
LIN {X 0,Y 164.338,Z 266.496,A -85,B 0,C 180,E1 -23336.139,E2 -23336.139} C_VEL
LIN {X 0,Y 164.331,Z 266.491,A -85,B 0,C 180,E1 -23341.239,E2 -23341.239} C_VEL
LIN {X 0,Y 164.309,Z 266.514,A -85,B 0,C 180,E1 -23346.79,E2 -23346.79} C_VEL
LIN {X 0,Y 164.334,Z 266.505,A -85,B 0,C 180,E1 -23349.909,E2 -23349.909} C_VEL
LIN {X 0,Y 164.351,Z 266.511,A -85,B 0,C 180,E1 -23353.396,E2 -23353.396} C_VEL
LIN {X 0,Y 164.366,Z 266.496,A -85,B 0,C 180,E1 -23356.859,E2 -23356.859} C_VEL
LIN {X 0,Y 164.354,Z 266.511,A -85,B 0,C 180,E1 -23360.333,E2 -23360.333} C_VEL
LIN {X 0,Y 164.331,Z 266.501,A -85,B 0,C 180,E1 -23364.355,E2 -23364.355} C_VEL
LIN {X 0,Y 164.371,Z 266.51,A -85,B 0,C 180,E1 -23369.152,E2 -23369.152} C_VEL
LIN {X 0,Y 164.392,Z 266.49,A -85,B 0,C 180,E1 -23374.71,E2 -23374.71} C_VEL
LIN {X 0,Y 164.409,Z 266.503,A -85,B 0,C 180,E1 -23380.134,E2 -23380.134} C_VEL
LIN {X 0,Y 164.482,Z 266.482,A -85,B 0,C 180,E1 -23385.163,E2 -23385.163} C_VEL
LIN {X 0,Y 164.765,Z 266.456,A -85,B 0,C 180,E1 -23390.193,E2 -23390.193} C_VEL
LIN {X 0,Y 164.824,Z 266.436,A -85,B 0,C 180,E1 -23392.667,E2 -23392.667} C_VEL
LIN {X 0,Y 165.282,Z 266.387,A -85,B 0,C 180,E1 -23400.016,E2 -23400.016} C_VEL
LIN {X 0,Y 164.832,Z 266.411,A -85,B 0,C 180,E1 -23407.365,E2 -23407.365} C_VEL
LIN {X 0,Y 164.719,Z 266.465,A -85,B 0,C 180,E1 -23411.072,E2 -23411.072} C_VEL
LIN {X 0,Y 164.457,Z 266.467,A -85,B 0,C 180,E1 -23417.422,E2 -23417.422} C_VEL
LIN {X 0,Y 164.376,Z 266.505,A -85,B 0,C 180,E1 -23422.647,E2 -23422.647} C_VEL
LIN {X 0,Y 164.396,Z 266.499,A -85,B 0,C 180,E1 -23426.127,E2 -23426.127} C_VEL
LIN {X 0,Y 164.386,Z 266.5,A -85,B 0,C 180,E1 -23431.227,E2 -23431.227} C_VEL
LIN {X 0,Y 164.31,Z 266.499,A -85,B 0,C 180,E1 -23436.803,E2 -23436.803} C_VEL
LIN {X 0,Y 164.315,Z 266.517,A -85,B 0,C 180,E1 -23439.927,E2 -23439.927} C_VEL
LIN {X 0,Y 164.283,Z 266.511,A -85,B 0,C 180,E1 -23443.338,E2 -23443.338} C_VEL
LIN {X 0,Y 164.36,Z 266.729,A -85,B 0,C 180,E1 -23447.879,E2 -23447.879} C_VEL
LIN {X 0,Y 164.655,Z 267.96,A -85,B 0,C 180,E1 -23448.345,E2 -23448.345} C_VEL
LIN {X 0,Y 168.172,Z 275.24,A -85,B 0,C 180,E1 -23449.489,E2 -23449.489} C_VEL
LIN {X 0,Y 174.626,Z 291.085,A -85,B 0,C 180,E1 -23451.569,E2 -23451.569} C_VEL
LIN {X 0,Y 181.785,Z 311.352,A -85,B 0,C 180,E1 -23453.828,E2 -23453.828} C_VEL
LIN {X 0,Y 182.946,Z 321.268,A -85,B 0,C 180,E1 -23454.52,E2 -23454.52} C_VEL
LIN {X 0,Y 179.908,Z 372.504,A -85,B 0,C 180,E1 -23456.778,E2 -23456.778} C_VEL
LIN {X 0,Y 178.713,Z 385.55,A -85,B 0,C 180,E1 -23457.68,E2 -23457.68} C_VEL
LIN {X 0,Y 177.022,Z 397.757,A -85,B 0,C 180,E1 -23458.924,E2 -23458.924} C_VEL
LIN {X 0,Y 174.952,Z 409.374,A -85,B 0,C 180,E1 -23460.518,E2 -23460.518} C_VEL
LIN {X 0,Y 172.825,Z 420.131,A -85,B 0,C 180,E1 -23462.443,E2 -23462.443} C_VEL
LIN {X 0,Y 170.605,Z 430.082,A -85,B 0,C 180,E1 -23464.694,E2 -23464.694} C_VEL
LIN {X 0,Y 168.321,Z 439.664,A -85,B 0,C 180,E1 -23467.419,E2 -23467.419} C_VEL
LIN {X 0,Y 167.935,Z 441.504,A -85,B 0,C 180,E1 -23468.021,E2 -23468.021} C_VEL
LIN {X 0,Y 166.245,Z 445.543,A -85,B 0,C 180,E1 -23469.386,E2 -23469.386} C_VEL
LIN {X 0,Y 161.881,Z 451.594,A -85,B 0,C 180,E1 -23471.677,E2 -23471.677} C_VEL
LIN {X 0,Y 157.736,Z 457.031,A -85,B 0,C 180,E1 -23474.261,E2 -23474.261} C_VEL
LIN {X 0,Y 156.432,Z 460.107,A -85,B 0,C 180,E1 -23476.043,E2 -23476.043} C_VEL
LIN {X 0,Y 155.469,Z 465.343,A -85,B 0,C 180,E1 -23479.578,E2 -23479.578} C_VEL
LIN {X 0,Y 154.88,Z 469.863,A -85,B 0,C 180,E1 -23483.482,E2 -23483.482} C_VEL
LIN {X 0,Y 154.694,Z 473.251,A -85,B 0,C 180,E1 -23487.392,E2 -23487.392} C_VEL
LIN {X 0,Y 154.685,Z 475.563,A -85,B 0,C 180,E1 -23491.201,E2 -23491.201} C_VEL
LIN {X 0,Y 154.748,Z 476.996,A -85,B 0,C 180,E1 -23495.207,E2 -23495.207} C_VEL
LIN {X 0,Y 155.618,Z 477.434,A -85,B 0,C 180,E1 -23500.403,E2 -23500.403} C_VEL
LIN {X 0,Y 157.507,Z 476.365,A -85,B 0,C 180,E1 -23505.524,E2 -23505.524} C_VEL
LIN {X 0,Y 158.842,Z 475.26,A -85,B 0,C 180,E1 -23508.037,E2 -23508.037} C_VEL
LIN {X 0,Y 160.54,Z 473.726,A -85,B 0,C 180,E1 -23510.496,E2 -23510.496} C_VEL
LIN {X 0,Y 163.799,Z 470.666,A -85,B 0,C 180,E1 -23514.05,E2 -23514.05} C_VEL
LIN {X 0,Y 167.686,Z 466.611,A -85,B 0,C 180,E1 -23517.448,E2 -23517.448} C_VEL
LIN {X 0,Y 172.586,Z 460.611,A -85,B 0,C 180,E1 -23521.2,E2 -23521.2} C_VEL
LIN {X 0,Y 177.603,Z 453.909,A -85,B 0,C 180,E1 -23524.32,E2 -23524.32} C_VEL
LIN {X 0,Y 183.205,Z 445.765,A -85,B 0,C 180,E1 -23527.165,E2 -23527.165} C_VEL
LIN {X 0,Y 188.258,Z 437.492,A -85,B 0,C 180,E1 -23529.388,E2 -23529.388} C_VEL
LIN {X 0,Y 193.554,Z 427.485,A -85,B 0,C 180,E1 -23531.498,E2 -23531.498} C_VEL
LIN {X 0,Y 198.024,Z 417.734,A -85,B 0,C 180,E1 -23533.088,E2 -23533.088} C_VEL
LIN {X 0,Y 202.682,Z 405.624,A -85,B 0,C 180,E1 -23534.596,E2 -23534.596} C_VEL
LIN {X 0,Y 206.339,Z 393.81,A -85,B 0,C 180,E1 -23535.66,E2 -23535.66} C_VEL
LIN {X 0,Y 209.392,Z 380.649,A -85,B 0,C 180,E1 -23536.498,E2 -23536.498} C_VEL
LIN {X 0,Y 211.489,Z 366.567,A -85,B 0,C 180,E1 -23537.103,E2 -23537.103} C_VEL
LIN {X 0,Y 213.93,Z 343.262,A -85,B 0,C 180,E1 -23537.945,E2 -23537.945} C_VEL
LIN {X 0,Y 211.518,Z 336.645,A -85,B 0,C 180,E1 -23539.959,E2 -23539.959} C_VEL
LIN {X 0,Y 208.798,Z 330.217,A -85,B 0,C 180,E1 -23542.43,E2 -23542.43} C_VEL
LIN {X 0,Y 206.887,Z 326.151,A -85,B 0,C 180,E1 -23544.437,E2 -23544.437} C_VEL
LIN {X 0,Y 204.924,Z 322.089,A -85,B 0,C 180,E1 -23546.87,E2 -23546.87} C_VEL
LIN {X 0,Y 202.775,Z 317.798,A -85,B 0,C 180,E1 -23550.39,E2 -23550.39} C_VEL
LIN {X 0,Y 201.036,Z 314.626,A -85,B 0,C 180,E1 -23555.87,E2 -23555.87} C_VEL
LIN {X 0,Y 200.886,Z 314.308,A -85,B 0,C 180,E1 -23557.354,E2 -23557.354} C_VEL
LIN {X 0,Y 201.345,Z 314.844,A -85,B 0,C 180,E1 -23561.9,E2 -23561.9} C_VEL
LIN {X 0,Y 203.628,Z 317.907,A -85,B 0,C 180,E1 -23567.121,E2 -23567.121} C_VEL
LIN {X 0,Y 205.913,Z 322.095,A -85,B 0,C 180,E1 -23570.414,E2 -23570.414} C_VEL
LIN {X 0,Y 208.443,Z 326.377,A -85,B 0,C 180,E1 -23573.101,E2 -23573.101} C_VEL
LIN {X 0,Y 211.518,Z 333.436,A -85,B 0,C 180,E1 -23575.983,E2 -23575.983} C_VEL
LIN {X 0,Y 213.568,Z 338.267,A -85,B 0,C 180,E1 -23577.656,E2 -23577.656} C_VEL
LIN {X 0,Y 214.172,Z 340.051,A -85,B 0,C 180,E1 -23578.158,E2 -23578.158} C_VEL
LIN {X 0,Y 210.519,Z 372.724,A -85,B 0,C 180,E1 -23579.389,E2 -23579.389} C_VEL
LIN {X 0,Y 208.02,Z 385.481,A -85,B 0,C 180,E1 -23580.1,E2 -23580.1} C_VEL
LIN {X 0,Y 204.927,Z 397.024,A -85,B 0,C 180,E1 -23581.018,E2 -23581.018} C_VEL
LIN {X 0,Y 200.842,Z 409.084,A -85,B 0,C 180,E1 -23582.368,E2 -23582.368} C_VEL
LIN {X 0,Y 195.898,Z 420.842,A -85,B 0,C 180,E1 -23584.101,E2 -23584.101} C_VEL
LIN {X 0,Y 190.812,Z 430.977,A -85,B 0,C 180,E1 -23586.073,E2 -23586.073} C_VEL
LIN {X 0,Y 184.768,Z 441.316,A -85,B 0,C 180,E1 -23588.736,E2 -23588.736} C_VEL
LIN {X 0,Y 179.288,Z 449.507,A -85,B 0,C 180,E1 -23591.506,E2 -23591.506} C_VEL
LIN {X 0,Y 174.183,Z 456.191,A -85,B 0,C 180,E1 -23594.47,E2 -23594.47} C_VEL
LIN {X 0,Y 169.625,Z 461.626,A -85,B 0,C 180,E1 -23597.662,E2 -23597.662} C_VEL
LIN {X 0,Y 165.622,Z 465.926,A -85,B 0,C 180,E1 -23601.019,E2 -23601.019} C_VEL
LIN {X 0,Y 162.188,Z 469.212,A -85,B 0,C 180,E1 -23604.509,E2 -23604.509} C_VEL
LIN {X 0,Y 158.821,Z 471.971,A -85,B 0,C 180,E1 -23609.107,E2 -23609.107} C_VEL
LIN {X 0,Y 157.005,Z 473.106,A -85,B 0,C 180,E1 -23612.468,E2 -23612.468} C_VEL
LIN {X 0,Y 155.631,Z 473.512,A -85,B 0,C 180,E1 -23615.924,E2 -23615.924} C_VEL
LIN {X 0,Y 154.788,Z 473.206,A -85,B 0,C 180,E1 -23619.486,E2 -23619.486} C_VEL
LIN {X 0,Y 154.265,Z 472.118,A -85,B 0,C 180,E1 -23623.211,E2 -23623.211} C_VEL
LIN {X 0,Y 154.152,Z 470.247,A -85,B 0,C 180,E1 -23626.86,E2 -23626.86} C_VEL
LIN {X 0,Y 154.42,Z 467.381,A -85,B 0,C 180,E1 -23630.656,E2 -23630.656} C_VEL
LIN {X 0,Y 155.101,Z 463.327,A -85,B 0,C 180,E1 -23634.614,E2 -23634.614} C_VEL
LIN {X 0,Y 156.188,Z 457.798,A -85,B 0,C 180,E1 -23638.714,E2 -23638.714} C_VEL
LIN {X 0,Y 157.836,Z 450.432,A -85,B 0,C 180,E1 -23642.897,E2 -23642.897} C_VEL
LIN {X 0,Y 159.989,Z 441.814,A -85,B 0,C 180,E1 -23646.717,E2 -23646.717} C_VEL
LIN {X 0,Y 162.389,Z 431.936,A -85,B 0,C 180,E1 -23650.12,E2 -23650.12} C_VEL
LIN {X 0,Y 164.966,Z 421.434,A -85,B 0,C 180,E1 -23652.959,E2 -23652.959} C_VEL
LIN {X 0,Y 167.479,Z 409.703,A -85,B 0,C 180,E1 -23655.422,E2 -23655.422} C_VEL
LIN {X 0,Y 169.867,Z 396.894,A -85,B 0,C 180,E1 -23657.459,E2 -23657.459} C_VEL
LIN {X 0,Y 171.729,Z 384.076,A -85,B 0,C 180,E1 -23658.945,E2 -23658.945} C_VEL
LIN {X 0,Y 173.259,Z 370.482,A -85,B 0,C 180,E1 -23660.007,E2 -23660.007} C_VEL
LIN {X 0,Y 176.816,Z 314.094,A -85,B 0,C 180,E1 -23662.6,E2 -23662.6} C_VEL
LIN {X 0,Y 170.402,Z 295.301,A -85,B 0,C 180,E1 -23664.717,E2 -23664.717} C_VEL
LIN {X 0,Y 166.146,Z 284.423,A -85,B 0,C 180,E1 -23666.139,E2 -23666.139} C_VEL
LIN {X 0,Y 158.351,Z 268.625,A -85,B 0,C 180,E1 -23668.732,E2 -23668.732} C_VEL
LIN {X 0,Y 158.11,Z 267.41,A -85,B 0,C 180,E1 -23669.287,E2 -23669.287} C_VEL
LIN {X 0,Y 158.202,Z 267.268,A -85,B 0,C 180,E1 -23670.004,E2 -23670.004} C_VEL
LIN {X 0,Y 157.668,Z 267.332,A -85,B 0,C 180,E1 -23675.119,E2 -23675.119} C_VEL
LIN {X 0,Y 157.744,Z 267.335,A -85,B 0,C 180,E1 -23677.685,E2 -23677.685} C_VEL
LIN {X 0,Y 157.615,Z 267.333,A -85,B 0,C 180,E1 -23681.302,E2 -23681.302} C_VEL
LIN {X 0,Y 157.383,Z 267.373,A -85,B 0,C 180,E1 -23685.546,E2 -23685.546} C_VEL
LIN {X 0,Y 157.318,Z 267.378,A -85,B 0,C 180,E1 -23690.944,E2 -23690.944} C_VEL
LIN {X 0,Y 157.265,Z 267.365,A -85,B 0,C 180,E1 -23696.693,E2 -23696.693} C_VEL
LIN {X 0,Y 157.235,Z 267.386,A -85,B 0,C 180,E1 -23702.442,E2 -23702.442} C_VEL
LIN {X 0,Y 157.283,Z 267.39,A -85,B 0,C 180,E1 -23706.49,E2 -23706.49} C_VEL
LIN {X 0,Y 157.257,Z 267.396,A -85,B 0,C 180,E1 -23712.101,E2 -23712.101} C_VEL
LIN {X 0,Y 157.281,Z 267.382,A -85,B 0,C 180,E1 -23715.645,E2 -23715.645} C_VEL
LIN {X 0,Y 157.27,Z 267.393,A -85,B 0,C 180,E1 -23721.297,E2 -23721.297} C_VEL
LIN {X 0,Y 157.278,Z 267.378,A -85,B 0,C 180,E1 -23724.509,E2 -23724.509} C_VEL
LIN {X 0,Y 157.275,Z 267.39,A -85,B 0,C 180,E1 -23728.114,E2 -23728.114} C_VEL
LIN {X 0,Y 157.3,Z 267.376,A -85,B 0,C 180,E1 -23733.483,E2 -23733.483} C_VEL
LIN {X 0,Y 157.352,Z 267.383,A -85,B 0,C 180,E1 -23739.72,E2 -23739.72} C_VEL
LIN {X 0,Y 157.413,Z 267.359,A -85,B 0,C 180,E1 -23744.48,E2 -23744.48} C_VEL
LIN {X 0,Y 157.688,Z 267.34,A -85,B 0,C 180,E1 -23749.748,E2 -23749.748} C_VEL
LIN {X 0,Y 157.762,Z 267.316,A -85,B 0,C 180,E1 -23752.337,E2 -23752.337} C_VEL
LIN {X 0,Y 158.245,Z 267.263,A -85,B 0,C 180,E1 -23760.017,E2 -23760.017} C_VEL
LIN {X 0,Y 157.771,Z 267.292,A -85,B 0,C 180,E1 -23767.696,E2 -23767.696} C_VEL
LIN {X 0,Y 157.65,Z 267.346,A -85,B 0,C 180,E1 -23771.24,E2 -23771.24} C_VEL
LIN {X 0,Y 157.435,Z 267.359,A -85,B 0,C 180,E1 -23775.552,E2 -23775.552} C_VEL
LIN {X 0,Y 157.334,Z 267.363,A -85,B 0,C 180,E1 -23780.954,E2 -23780.954} C_VEL
LIN {X 0,Y 157.337,Z 267.372,A -85,B 0,C 180,E1 -23786.693,E2 -23786.693} C_VEL
LIN {X 0,Y 157.297,Z 267.391,A -85,B 0,C 180,E1 -23792.44,E2 -23792.44} C_VEL
LIN {X 0,Y 157.289,Z 267.372,A -85,B 0,C 180,E1 -23796.453,E2 -23796.453} C_VEL
LIN {X 0,Y 157.22,Z 267.386,A -85,B 0,C 180,E1 -23802.127,E2 -23802.127} C_VEL
LIN {X 0,Y 157.265,Z 267.62,A -85,B 0,C 180,E1 -23806.425,E2 -23806.425} C_VEL
LIN {X 0,Y 157.609,Z 268.855,A -85,B 0,C 180,E1 -23806.932,E2 -23806.932} C_VEL
LIN {X 0,Y 162.325,Z 278.186,A -85,B 0,C 180,E1 -23808.532,E2 -23808.532} C_VEL
LIN {X 0,Y 168.626,Z 293.822,A -85,B 0,C 180,E1 -23810.667,E2 -23810.667} C_VEL
LIN {X 0,Y 175.672,Z 313.789,A -85,B 0,C 180,E1 -23812.99,E2 -23812.99} C_VEL
LIN {X 0,Y 176.531,Z 321.901,A -85,B 0,C 180,E1 -23813.569,E2 -23813.569} C_VEL
LIN {X 0,Y 173.291,Z 373.641,A -85,B 0,C 180,E1 -23815.928,E2 -23815.928} C_VEL
LIN {X 0,Y 171.928,Z 387.026,A -85,B 0,C 180,E1 -23816.94,E2 -23816.94} C_VEL
LIN {X 0,Y 170.034,Z 399.937,A -85,B 0,C 180,E1 -23818.367,E2 -23818.367} C_VEL
LIN {X 0,Y 167.704,Z 411.806,A -85,B 0,C 180,E1 -23820.151,E2 -23820.151} C_VEL
LIN {X 0,Y 165.238,Z 423.314,A -85,B 0,C 180,E1 -23822.445,E2 -23822.445} C_VEL
LIN {X 0,Y 163.014,Z 433.02,A -85,B 0,C 180,E1 -23824.903,E2 -23824.903} C_VEL
LIN {X 0,Y 160.978,Z 441.428,A -85,B 0,C 180,E1 -23827.538,E2 -23827.538} C_VEL
LIN {X 0,Y 158.934,Z 449.464,A -85,B 0,C 180,E1 -23830.627,E2 -23830.627} C_VEL
LIN {X 0,Y 156.976,Z 457.276,A -85,B 0,C 180,E1 -23834.413,E2 -23834.413} C_VEL
LIN {X 0,Y 156.432,Z 460.107,A -85,B 0,C 180,E1 -23836.043,E2 -23836.043} C_VEL
LIN {X 0,Y 155.231,Z 462.989,A -85,B 0,C 180,E1 -23837.895,E2 -23837.895} C_VEL
LIN {X 0,Y 151.662,Z 467.032,A -85,B 0,C 180,E1 -23841.004,E2 -23841.004} C_VEL
LIN {X 0,Y 148.866,Z 469.767,A -85,B 0,C 180,E1 -23843.663,E2 -23843.663} C_VEL
LIN {X 0,Y 147.691,Z 471.626,A -85,B 0,C 180,E1 -23845.802,E2 -23845.802} C_VEL
LIN {X 0,Y 147.595,Z 472.2,A -85,B 0,C 180,E1 -23846.537,E2 -23846.537} C_VEL
LIN {X 0,Y 147.632,Z 474.842,A -85,B 0,C 180,E1 -23850.608,E2 -23850.608} C_VEL
LIN {X 0,Y 147.673,Z 476.725,A -85,B 0,C 180,E1 -23855.457,E2 -23855.457} C_VEL
LIN {X 0,Y 148.011,Z 477.249,A -85,B 0,C 180,E1 -23858.185,E2 -23858.185} C_VEL
LIN {X 0,Y 148.624,Z 477.369,A -85,B 0,C 180,E1 -23860.898,E2 -23860.898} C_VEL
LIN {X 0,Y 150.657,Z 476.439,A -85,B 0,C 180,E1 -23866.249,E2 -23866.249} C_VEL
LIN {X 0,Y 153.92,Z 474.012,A -85,B 0,C 180,E1 -23871.42,E2 -23871.42} C_VEL
LIN {X 0,Y 157.357,Z 471.103,A -85,B 0,C 180,E1 -23875.101,E2 -23875.101} C_VEL
LIN {X 0,Y 161.439,Z 467.21,A -85,B 0,C 180,E1 -23878.606,E2 -23878.606} C_VEL
LIN {X 0,Y 166.58,Z 461.485,A -85,B 0,C 180,E1 -23882.433,E2 -23882.433} C_VEL
LIN {X 0,Y 172.758,Z 453.761,A -85,B 0,C 180,E1 -23886.143,E2 -23886.143} C_VEL
LIN {X 0,Y 178.69,Z 445.664,A -85,B 0,C 180,E1 -23888.992,E2 -23888.992} C_VEL
LIN {X 0,Y 184.021,Z 437.428,A -85,B 0,C 180,E1 -23891.203,E2 -23891.203} C_VEL
LIN {X 0,Y 189.549,Z 427.426,A -85,B 0,C 180,E1 -23893.303,E2 -23893.303} C_VEL
LIN {X 0,Y 194.231,Z 417.66,A -85,B 0,C 180,E1 -23894.871,E2 -23894.871} C_VEL
LIN {X 0,Y 199.054,Z 405.567,A -85,B 0,C 180,E1 -23896.363,E2 -23896.363} C_VEL
LIN {X 0,Y 202.975,Z 393.484,A -85,B 0,C 180,E1 -23897.422,E2 -23897.422} C_VEL
LIN {X 0,Y 206.023,Z 380.919,A -85,B 0,C 180,E1 -23898.213,E2 -23898.213} C_VEL
LIN {X 0,Y 208.234,Z 366.984,A -85,B 0,C 180,E1 -23898.816,E2 -23898.816} C_VEL
LIN {X 0,Y 210.513,Z 346.627,A -85,B 0,C 180,E1 -23899.534,E2 -23899.534} C_VEL
LIN {X 0,Y 208.077,Z 339.815,A -85,B 0,C 180,E1 -23901.785,E2 -23901.785} C_VEL
LIN {X 0,Y 205.667,Z 333.921,A -85,B 0,C 180,E1 -23904.38,E2 -23904.38} C_VEL
LIN {X 0,Y 203.356,Z 328.785,A -85,B 0,C 180,E1 -23907.392,E2 -23907.392} C_VEL
LIN {X 0,Y 201.358,Z 324.494,A -85,B 0,C 180,E1 -23910.975,E2 -23910.975} C_VEL
LIN {X 0,Y 199.9,Z 321.602,A -85,B 0,C 180,E1 -23916.068,E2 -23916.068} C_VEL
LIN {X 0,Y 199.813,Z 321.401,A -85,B 0,C 180,E1 -23919.394,E2 -23919.394} C_VEL
LIN {X 0,Y 200.36,Z 322.145,A -85,B 0,C 180,E1 -23922.462,E2 -23922.462} C_VEL
LIN {X 0,Y 202.203,Z 324.677,A -85,B 0,C 180,E1 -23926.687,E2 -23926.687} C_VEL
LIN {X 0,Y 204.284,Z 328.759,A -85,B 0,C 180,E1 -23929.87,E2 -23929.87} C_VEL
LIN {X 0,Y 206.592,Z 332.958,A -85,B 0,C 180,E1 -23932.515,E2 -23932.515} C_VEL
LIN {X 0,Y 210.026,Z 341.319,A -85,B 0,C 180,E1 -23935.896,E2 -23935.896} C_VEL
LIN {X 0,Y 210.763,Z 343.351,A -85,B 0,C 180,E1 -23936.55,E2 -23936.55} C_VEL
LIN {X 0,Y 207.358,Z 372.268,A -85,B 0,C 180,E1 -23937.632,E2 -23937.632} C_VEL
LIN {X 0,Y 204.659,Z 385.554,A -85,B 0,C 180,E1 -23938.355,E2 -23938.355} C_VEL
LIN {X 0,Y 201.093,Z 398.13,A -85,B 0,C 180,E1 -23939.364,E2 -23939.364} C_VEL
LIN {X 0,Y 196.784,Z 410.074,A -85,B 0,C 180,E1 -23940.715,E2 -23940.715} C_VEL
LIN {X 0,Y 192.048,Z 420.876,A -85,B 0,C 180,E1 -23942.312,E2 -23942.312} C_VEL
LIN {X 0,Y 186.632,Z 431.204,A -85,B 0,C 180,E1 -23944.305,E2 -23944.305} C_VEL
LIN {X 0,Y 180.848,Z 440.597,A -85,B 0,C 180,E1 -23946.68,E2 -23946.68} C_VEL
LIN {X 0,Y 174.594,Z 449.487,A -85,B 0,C 180,E1 -23949.671,E2 -23949.671} C_VEL
LIN {X 0,Y 168.576,Z 456.854,A -85,B 0,C 180,E1 -23953.02,E2 -23953.02} C_VEL
LIN {X 0,Y 163.984,Z 461.942,A -85,B 0,C 180,E1 -23956.102,E2 -23956.102} C_VEL
LIN {X 0,Y 160.071,Z 465.862,A -85,B 0,C 180,E1 -23959.207,E2 -23959.207} C_VEL
LIN {X 0,Y 156.703,Z 468.865,A -85,B 0,C 180,E1 -23962.408,E2 -23962.408} C_VEL
LIN {X 0,Y 154.674,Z 470.499,A -85,B 0,C 180,E1 -23964.679,E2 -23964.679} C_VEL
LIN {X 0,Y 151.939,Z 472.392,A -85,B 0,C 180,E1 -23968.507,E2 -23968.507} C_VEL
LIN {X 0,Y 149.834,Z 473.409,A -85,B 0,C 180,E1 -23972.413,E2 -23972.413} C_VEL
LIN {X 0,Y 147.915,Z 473.399,A -85,B 0,C 180,E1 -23978.121,E2 -23978.121} C_VEL
LIN {X 0,Y 147.298,Z 472.456,A -85,B 0,C 180,E1 -23981.883,E2 -23981.883} C_VEL
LIN {X 0,Y 147.045,Z 470.659,A -85,B 0,C 180,E1 -23985.771,E2 -23985.771} C_VEL
LIN {X 0,Y 147.221,Z 467.934,A -85,B 0,C 180,E1 -23989.768,E2 -23989.768} C_VEL
LIN {X 0,Y 147.851,Z 464.089,A -85,B 0,C 180,E1 -23993.873,E2 -23993.873} C_VEL
LIN {X 0,Y 148.86,Z 458.788,A -85,B 0,C 180,E1 -23998.152,E2 -23998.152} C_VEL
LIN {X 0,Y 150.496,Z 451.807,A -85,B 0,C 180,E1 -24002.487,E2 -24002.487} C_VEL
LIN {X 0,Y 152.366,Z 444.1,A -85,B 0,C 180,E1 -24006.223,E2 -24006.223} C_VEL
LIN {X 0,Y 154.921,Z 434.274,A -85,B 0,C 180,E1 -24009.974,E2 -24009.974} C_VEL
LIN {X 0,Y 157.644,Z 423.449,A -85,B 0,C 180,E1 -24013.16,E2 -24013.16} C_VEL
LIN {X 0,Y 160.218,Z 412.449,A -85,B 0,C 180,E1 -24015.682,E2 -24015.682} C_VEL
LIN {X 0,Y 162.515,Z 400.887,A -85,B 0,C 180,E1 -24017.741,E2 -24017.741} C_VEL
LIN {X 0,Y 164.658,Z 387.925,A -85,B 0,C 180,E1 -24019.447,E2 -24019.447} C_VEL
LIN {X 0,Y 166.255,Z 375.038,A -85,B 0,C 180,E1 -24020.651,E2 -24020.651} C_VEL
LIN {X 0,Y 167.505,Z 360.421,A -85,B 0,C 180,E1 -24021.477,E2 -24021.477} C_VEL
LIN {X 0,Y 170.224,Z 315.201,A -85,B 0,C 180,E1 -24023.606,E2 -24023.606} C_VEL
LIN {X 0,Y 163.96,Z 296.706,A -85,B 0,C 180,E1 -24025.818,E2 -24025.818} C_VEL
LIN {X 0,Y 160.388,Z 287.676,A -85,B 0,C 180,E1 -24027.066,E2 -24027.066} C_VEL
LIN {X 0,Y 151.409,Z 269.476,A -85,B 0,C 180,E1 -24030.254,E2 -24030.254} C_VEL
LIN {X 0,Y 151.07,Z 268.307,A -85,B 0,C 180,E1 -24030.838,E2 -24030.838} C_VEL
LIN {X 0,Y 150.679,Z 268.21,A -85,B 0,C 180,E1 -24038.048,E2 -24038.048} C_VEL
LIN {X 0,Y 150.549,Z 268.214,A -85,B 0,C 180,E1 -24041.49,E2 -24041.49} C_VEL
LIN {X 0,Y 150.295,Z 268.245,A -85,B 0,C 180,E1 -24046.299,E2 -24046.299} C_VEL
LIN {X 0,Y 150.3,Z 268.249,A -85,B 0,C 180,E1 -24050.801,E2 -24050.801} C_VEL
LIN {X 0,Y 150.197,Z 268.237,A -85,B 0,C 180,E1 -24057.292,E2 -24057.292} C_VEL
LIN {X 0,Y 150.175,Z 268.266,A -85,B 0,C 180,E1 -24062.647,E2 -24062.647} C_VEL
LIN {X 0,Y 150.195,Z 268.268,A -85,B 0,C 180,E1 -24067.472,E2 -24067.472} C_VEL
LIN {X 0,Y 150.197,Z 268.274,A -85,B 0,C 180,E1 -24071.556,E2 -24071.556} C_VEL
LIN {X 0,Y 150.256,Z 268.257,A -85,B 0,C 180,E1 -24075.473,E2 -24075.473} C_VEL
LIN {X 0,Y 150.213,Z 268.269,A -85,B 0,C 180,E1 -24079.106,E2 -24079.106} C_VEL
LIN {X 0,Y 150.22,Z 268.267,A -85,B 0,C 180,E1 -24082.694,E2 -24082.694} C_VEL
LIN {X 0,Y 150.2,Z 268.266,A -85,B 0,C 180,E1 -24087.384,E2 -24087.384} C_VEL
LIN {X 0,Y 150.227,Z 268.261,A -85,B 0,C 180,E1 -24092.74,E2 -24092.74} C_VEL
LIN {X 0,Y 150.277,Z 268.266,A -85,B 0,C 180,E1 -24099.294,E2 -24099.294} C_VEL
LIN {X 0,Y 150.316,Z 268.242,A -85,B 0,C 180,E1 -24103.728,E2 -24103.728} C_VEL
LIN {X 0,Y 150.608,Z 268.224,A -85,B 0,C 180,E1 -24109.261,E2 -24109.261} C_VEL
LIN {X 0,Y 150.684,Z 268.199,A -85,B 0,C 180,E1 -24111.975,E2 -24111.975} C_VEL
LIN {X 0,Y 151.205,Z 268.14,A -85,B 0,C 180,E1 -24120.018,E2 -24120.018} C_VEL
LIN {X 0,Y 150.695,Z 268.176,A -85,B 0,C 180,E1 -24128.06,E2 -24128.06} C_VEL
LIN {X 0,Y 150.592,Z 268.225,A -85,B 0,C 180,E1 -24131.444,E2 -24131.444} C_VEL
LIN {X 0,Y 150.34,Z 268.233,A -85,B 0,C 180,E1 -24136.306,E2 -24136.306} C_VEL
LIN {X 0,Y 150.308,Z 268.233,A -85,B 0,C 180,E1 -24140.738,E2 -24140.738} C_VEL
LIN {X 0,Y 150.266,Z 268.245,A -85,B 0,C 180,E1 -24147.289,E2 -24147.289} C_VEL
LIN {X 0,Y 150.238,Z 268.271,A -85,B 0,C 180,E1 -24152.638,E2 -24152.638} C_VEL
LIN {X 0,Y 150.2,Z 268.258,A -85,B 0,C 180,E1 -24157.484,E2 -24157.484} C_VEL
LIN {X 0,Y 150.163,Z 268.266,A -85,B 0,C 180,E1 -24161.504,E2 -24161.504} C_VEL
LIN {X 0,Y 150.157,Z 268.441,A -85,B 0,C 180,E1 -24164.751,E2 -24164.751} C_VEL
LIN {X 0,Y 150.494,Z 269.737,A -85,B 0,C 180,E1 -24165.34,E2 -24165.34} C_VEL
LIN {X 0,Y 155.631,Z 279.318,A -85,B 0,C 180,E1 -24167.192,E2 -24167.192} C_VEL
LIN {X 0,Y 161.718,Z 293.956,A -85,B 0,C 180,E1 -24169.372,E2 -24169.372} C_VEL
LIN {X 0,Y 168.661,Z 313.68,A -85,B 0,C 180,E1 -24171.827,E2 -24171.827} C_VEL
LIN {X 0,Y 169.6,Z 317.428,A -85,B 0,C 180,E1 -24172.202,E2 -24172.202} C_VEL
LIN {X 0,Y 170.1,Z 322.858,A -85,B 0,C 180,E1 -24172.594,E2 -24172.594} C_VEL
LIN {X 0,Y 166.713,Z 374.261,A -85,B 0,C 180,E1 -24175.032,E2 -24175.032} C_VEL
LIN {X 0,Y 165.207,Z 388.095,A -85,B 0,C 180,E1 -24176.146,E2 -24176.146} C_VEL
LIN {X 0,Y 163.278,Z 400.712,A -85,B 0,C 180,E1 -24177.628,E2 -24177.628} C_VEL
LIN {X 0,Y 160.51,Z 413.906,A -85,B 0,C 180,E1 -24179.761,E2 -24179.761} C_VEL
LIN {X 0,Y 158.012,Z 425.026,A -85,B 0,C 180,E1 -24182.155,E2 -24182.155} C_VEL
LIN {X 0,Y 155.645,Z 434.781,A -85,B 0,C 180,E1 -24184.843,E2 -24184.843} C_VEL
LIN {X 0,Y 153.414,Z 443.381,A -85,B 0,C 180,E1 -24187.789,E2 -24187.789} C_VEL
LIN {X 0,Y 151.102,Z 452.434,A -85,B 0,C 180,E1 -24191.698,E2 -24191.698} C_VEL
LIN {X 0,Y 149.37,Z 459.824,A -85,B 0,C 180,E1 -24195.796,E2 -24195.796} C_VEL
LIN {X 0,Y 148.213,Z 466.238,A -85,B 0,C 180,E1 -24200.442,E2 -24200.442} C_VEL
LIN {X 0,Y 147.704,Z 470.521,A -85,B 0,C 180,E1 -24204.535,E2 -24204.535} C_VEL
LIN {X 0,Y 147.595,Z 472.2,A -85,B 0,C 180,E1 -24206.537,E2 -24206.537} C_VEL
LIN {X 0,Y 146.896,Z 473.767,A -85,B 0,C 180,E1 -24208.733,E2 -24208.733} C_VEL
LIN {X 0,Y 145.283,Z 475.007,A -85,B 0,C 180,E1 -24210.927,E2 -24210.927} C_VEL
LIN {X 0,Y 141.709,Z 476.581,A -85,B 0,C 180,E1 -24215.473,E2 -24215.473} C_VEL
LIN {X 0,Y 140.943,Z 476.974,A -85,B 0,C 180,E1 -24217.879,E2 -24217.879} C_VEL
LIN {X 0,Y 140.994,Z 477.05,A -85,B 0,C 180,E1 -24218.69,E2 -24218.69} C_VEL
LIN {X 0,Y 142.581,Z 477.093,A -85,B 0,C 180,E1 -24224.263,E2 -24224.263} C_VEL
LIN {X 0,Y 145.364,Z 475.581,A -85,B 0,C 180,E1 -24229.776,E2 -24229.776} C_VEL
LIN {X 0,Y 149.681,Z 472.552,A -85,B 0,C 180,E1 -24234.992,E2 -24234.992} C_VEL
LIN {X 0,Y 153.801,Z 469.147,A -85,B 0,C 180,E1 -24238.667,E2 -24238.667} C_VEL
LIN {X 0,Y 159.259,Z 463.847,A -85,B 0,C 180,E1 -24242.788,E2 -24242.788} C_VEL
LIN {X 0,Y 165.278,Z 457.15,A -85,B 0,C 180,E1 -24246.529,E2 -24246.529} C_VEL
LIN {X 0,Y 171.248,Z 449.847,A -85,B 0,C 180,E1 -24249.497,E2 -24249.497} C_VEL
LIN {X 0,Y 176.58,Z 442.468,A -85,B 0,C 180,E1 -24251.804,E2 -24251.804} C_VEL
LIN {X 0,Y 182.26,Z 433.623,A -85,B 0,C 180,E1 -24253.948,E2 -24253.948} C_VEL
LIN {X 0,Y 187.567,Z 424.061,A -85,B 0,C 180,E1 -24255.768,E2 -24255.768} C_VEL
LIN {X 0,Y 193.163,Z 412.113,A -85,B 0,C 180,E1 -24257.451,E2 -24257.451} C_VEL
LIN {X 0,Y 197.619,Z 400.368,A -85,B 0,C 180,E1 -24258.695,E2 -24258.695} C_VEL
LIN {X 0,Y 201.419,Z 387.538,A -85,B 0,C 180,E1 -24259.651,E2 -24259.651} C_VEL
LIN {X 0,Y 204.36,Z 373.458,A -85,B 0,C 180,E1 -24260.362,E2 -24260.362} C_VEL
LIN {X 0,Y 207.179,Z 349.797,A -85,B 0,C 180,E1 -24261.258,E2 -24261.258} C_VEL
LIN {X 0,Y 204.953,Z 343.348,A -85,B 0,C 180,E1 -24263.683,E2 -24263.683} C_VEL
LIN {X 0,Y 203.07,Z 338.7,A -85,B 0,C 180,E1 -24265.98,E2 -24265.98} C_VEL
LIN {X 0,Y 201.573,Z 334.968,A -85,B 0,C 180,E1 -24268.287,E2 -24268.287} C_VEL
LIN {X 0,Y 200.008,Z 331.289,A -85,B 0,C 180,E1 -24271.449,E2 -24271.449} C_VEL
LIN {X 0,Y 198.738,Z 328.522,A -85,B 0,C 180,E1 -24276.511,E2 -24276.511} C_VEL
LIN {X 0,Y 198.878,Z 328.565,A -85,B 0,C 180,E1 -24280.641,E2 -24280.641} C_VEL
LIN {X 0,Y 199.725,Z 330.042,A -85,B 0,C 180,E1 -24283.882,E2 -24283.882} C_VEL
LIN {X 0,Y 200.862,Z 331.653,A -85,B 0,C 180,E1 -24286.372,E2 -24286.372} C_VEL
LIN {X 0,Y 202.653,Z 335.387,A -85,B 0,C 180,E1 -24289.294,E2 -24289.294} C_VEL
LIN {X 0,Y 204.657,Z 339.273,A -85,B 0,C 180,E1 -24291.795,E2 -24291.795} C_VEL
LIN {X 0,Y 207.501,Z 346.884,A -85,B 0,C 180,E1 -24294.907,E2 -24294.907} C_VEL
LIN {X 0,Y 204.256,Z 372.939,A -85,B 0,C 180,E1 -24295.868,E2 -24295.868} C_VEL
LIN {X 0,Y 201.51,Z 385.91,A -85,B 0,C 180,E1 -24296.568,E2 -24296.568} C_VEL
LIN {X 0,Y 197.955,Z 398.026,A -85,B 0,C 180,E1 -24297.516,E2 -24297.516} C_VEL
LIN {X 0,Y 193.54,Z 409.835,A -85,B 0,C 180,E1 -24298.816,E2 -24298.816} C_VEL
LIN {X 0,Y 188.177,Z 421.479,A -85,B 0,C 180,E1 -24300.52,E2 -24300.52} C_VEL
LIN {X 0,Y 182.867,Z 431.05,A -85,B 0,C 180,E1 -24302.352,E2 -24302.352} C_VEL
LIN {X 0,Y 176.331,Z 441.155,A -85,B 0,C 180,E1 -24304.906,E2 -24304.906} C_VEL
LIN {X 0,Y 170.188,Z 449.422,A -85,B 0,C 180,E1 -24307.689,E2 -24307.689} C_VEL
LIN {X 0,Y 164.489,Z 456.134,A -85,B 0,C 180,E1 -24310.698,E2 -24310.698} C_VEL
LIN {X 0,Y 159.261,Z 461.539,A -85,B 0,C 180,E1 -24313.894,E2 -24313.894} C_VEL
LIN {X 0,Y 154.608,Z 465.875,A -85,B 0,C 180,E1 -24317.349,E2 -24317.349} C_VEL
LIN {X 0,Y 149.551,Z 469.941,A -85,B 0,C 180,E1 -24322.062,E2 -24322.062} C_VEL
LIN {X 0,Y 146.631,Z 471.91,A -85,B 0,C 180,E1 -24325.533,E2 -24325.533} C_VEL
LIN {X 0,Y 144.303,Z 473.139,A -85,B 0,C 180,E1 -24329.122,E2 -24329.122} C_VEL
LIN {X 0,Y 142.406,Z 473.698,A -85,B 0,C 180,E1 -24332.977,E2 -24332.977} C_VEL
LIN {X 0,Y 141.04,Z 473.499,A -85,B 0,C 180,E1 -24337.138,E2 -24337.138} C_VEL
LIN {X 0,Y 140.276,Z 472.483,A -85,B 0,C 180,E1 -24341.286,E2 -24341.286} C_VEL
LIN {X 0,Y 139.969,Z 470.652,A -85,B 0,C 180,E1 -24345.343,E2 -24345.343} C_VEL
LIN {X 0,Y 140.079,Z 468.062,A -85,B 0,C 180,E1 -24349.297,E2 -24349.297} C_VEL
LIN {X 0,Y 140.612,Z 464.703,A -85,B 0,C 180,E1 -24353.153,E2 -24353.153} C_VEL
LIN {X 0,Y 141.575,Z 459.742,A -85,B 0,C 180,E1 -24357.514,E2 -24357.514} C_VEL
LIN {X 0,Y 143.12,Z 453.021,A -85,B 0,C 180,E1 -24362.069,E2 -24362.069} C_VEL
LIN {X 0,Y 145.066,Z 445.329,A -85,B 0,C 180,E1 -24366.139,E2 -24366.139} C_VEL
LIN {X 0,Y 147.445,Z 436.526,A -85,B 0,C 180,E1 -24369.789,E2 -24369.789} C_VEL
LIN {X 0,Y 149.945,Z 426.853,A -85,B 0,C 180,E1 -24372.971,E2 -24372.971} C_VEL
LIN {X 0,Y 152.655,Z 416.198,A -85,B 0,C 180,E1 -24375.722,E2 -24375.722} C_VEL
LIN {X 0,Y 155.206,Z 404.338,A -85,B 0,C 180,E1 -24378.083,E2 -24378.083} C_VEL
LIN {X 0,Y 157.332,Z 392.947,A -85,B 0,C 180,E1 -24379.806,E2 -24379.806} C_VEL
LIN {X 0,Y 159.227,Z 379.652,A -85,B 0,C 180,E1 -24381.278,E2 -24381.278} C_VEL
LIN {X 0,Y 160.723,Z 365.331,A -85,B 0,C 180,E1 -24382.269,E2 -24382.269} C_VEL
LIN {X 0,Y 163.906,Z 316.924,A -85,B 0,C 180,E1 -24384.611,E2 -24384.611} C_VEL
LIN {X 0,Y 156.86,Z 296.242,A -85,B 0,C 180,E1 -24387.249,E2 -24387.249} C_VEL
LIN {X 0,Y 153.837,Z 289.331,A -85,B 0,C 180,E1 -24388.335,E2 -24388.335} C_VEL
LIN {X 0,Y 146.014,Z 273.216,A -85,B 0,C 180,E1 -24391.278,E2 -24391.278} C_VEL
LIN {X 0,Y 144.33,Z 270.753,A -85,B 0,C 180,E1 -24391.902,E2 -24391.902} C_VEL
LIN {X 0,Y 143.9,Z 269.389,A -85,B 0,C 180,E1 -24392.454,E2 -24392.454} C_VEL
LIN {X 0,Y 143.829,Z 269.12,A -85,B 0,C 180,E1 -24392.806,E2 -24392.806} C_VEL
LIN {X 0,Y 143.599,Z 269.086,A -85,B 0,C 180,E1 -24398.448,E2 -24398.448} C_VEL
LIN {X 0,Y 143.48,Z 269.095,A -85,B 0,C 180,E1 -24401.69,E2 -24401.69} C_VEL
LIN {X 0,Y 143.234,Z 269.116,A -85,B 0,C 180,E1 -24407.126,E2 -24407.126} C_VEL
LIN {X 0,Y 143.227,Z 269.135,A -85,B 0,C 180,E1 -24411.263,E2 -24411.263} C_VEL
LIN {X 0,Y 143.144,Z 269.11,A -85,B 0,C 180,E1 -24417.948,E2 -24417.948} C_VEL
LIN {X 0,Y 143.127,Z 269.152,A -85,B 0,C 180,E1 -24423.45,E2 -24423.45} C_VEL
LIN {X 0,Y 143.089,Z 269.149,A -85,B 0,C 180,E1 -24429.686,E2 -24429.686} C_VEL
LIN {X 0,Y 143.134,Z 269.154,A -85,B 0,C 180,E1 -24433.432,E2 -24433.432} C_VEL
LIN {X 0,Y 143.142,Z 269.139,A -85,B 0,C 180,E1 -24437.438,E2 -24437.438} C_VEL
LIN {X 0,Y 143.147,Z 269.152,A -85,B 0,C 180,E1 -24441.777,E2 -24441.777} C_VEL
LIN {X 0,Y 143.167,Z 269.141,A -85,B 0,C 180,E1 -24447.342,E2 -24447.342} C_VEL
LIN {X 0,Y 143.173,Z 269.145,A -85,B 0,C 180,E1 -24452.085,E2 -24452.085} C_VEL
LIN {X 0,Y 143.218,Z 269.144,A -85,B 0,C 180,E1 -24458.818,E2 -24458.818} C_VEL
LIN {X 0,Y 143.253,Z 269.124,A -85,B 0,C 180,E1 -24462.901,E2 -24462.901} C_VEL
LIN {X 0,Y 143.534,Z 269.104,A -85,B 0,C 180,E1 -24468.725,E2 -24468.725} C_VEL
LIN {X 0,Y 143.61,Z 269.082,A -85,B 0,C 180,E1 -24471.577,E2 -24471.577} C_VEL
LIN {X 0,Y 144.164,Z 269.016,A -85,B 0,C 180,E1 -24480.018,E2 -24480.018} C_VEL
LIN {X 0,Y 143.621,Z 269.06,A -85,B 0,C 180,E1 -24488.46,E2 -24488.46} C_VEL
LIN {X 0,Y 143.518,Z 269.106,A -85,B 0,C 180,E1 -24491.633,E2 -24491.633} C_VEL
LIN {X 0,Y 143.279,Z 269.102,A -85,B 0,C 180,E1 -24497.134,E2 -24497.134} C_VEL
LIN {X 0,Y 143.25,Z 269.116,A -85,B 0,C 180,E1 -24501.214,E2 -24501.214} C_VEL
LIN {X 0,Y 143.211,Z 269.119,A -85,B 0,C 180,E1 -24507.943,E2 -24507.943} C_VEL
LIN {X 0,Y 143.168,Z 269.15,A -85,B 0,C 180,E1 -24513.427,E2 -24513.427} C_VEL
LIN {X 0,Y 143.082,Z 269.163,A -85,B 0,C 180,E1 -24519.704,E2 -24519.704} C_VEL
LIN {X 0,Y 143.066,Z 269.288,A -85,B 0,C 180,E1 -24522.988,E2 -24522.988} C_VEL
LIN {X 0,Y 143.348,Z 270.488,A -85,B 0,C 180,E1 -24523.608,E2 -24523.608} C_VEL
LIN {X 0,Y 149.91,Z 282.34,A -85,B 0,C 180,E1 -24526.087,E2 -24526.087} C_VEL
LIN {X 0,Y 155.92,Z 296.989,A -85,B 0,C 180,E1 -24528.386,E2 -24528.386} C_VEL
LIN {X 0,Y 162.856,Z 316.986,A -85,B 0,C 180,E1 -24530.988,E2 -24530.988} C_VEL
LIN {X 0,Y 163.703,Z 322.307,A -85,B 0,C 180,E1 -24531.46,E2 -24531.46} C_VEL
LIN {X 0,Y 160.394,Z 372.564,A -85,B 0,C 180,E1 -24533.924,E2 -24533.924} C_VEL
LIN {X 0,Y 159.046,Z 385.589,A -85,B 0,C 180,E1 -24534.934,E2 -24534.934} C_VEL
LIN {X 0,Y 157.096,Z 398.232,A -85,B 0,C 180,E1 -24536.38,E2 -24536.38} C_VEL
LIN {X 0,Y 154.771,Z 409.641,A -85,B 0,C 180,E1 -24538.133,E2 -24538.133} C_VEL
LIN {X 0,Y 152.064,Z 421.572,A -85,B 0,C 180,E1 -24540.585,E2 -24540.585} C_VEL
LIN {X 0,Y 149.215,Z 433.036,A -85,B 0,C 180,E1 -24543.678,E2 -24543.678} C_VEL
LIN {X 0,Y 146.841,Z 441.951,A -85,B 0,C 180,E1 -24546.738,E2 -24546.738} C_VEL
LIN {X 0,Y 144.362,Z 451.239,A -85,B 0,C 180,E1 -24550.811,E2 -24550.811} C_VEL
LIN {X 0,Y 142.494,Z 458.679,A -85,B 0,C 180,E1 -24554.988,E2 -24554.988} C_VEL
LIN {X 0,Y 141.495,Z 463.703,A -85,B 0,C 180,E1 -24558.536,E2 -24558.536} C_VEL
LIN {X 0,Y 140.769,Z 468.542,A -85,B 0,C 180,E1 -24562.825,E2 -24562.825} C_VEL
LIN {X 0,Y 140.523,Z 472.209,A -85,B 0,C 180,E1 -24567.128,E2 -24567.128} C_VEL
LIN {X 0,Y 140.596,Z 474.085,A -85,B 0,C 180,E1 -24569.995,E2 -24569.995} C_VEL
LIN {X 0,Y 140.521,Z 475.473,A -85,B 0,C 180,E1 -24572.862,E2 -24572.862} C_VEL
LIN {X 0,Y 140.994,Z 477.05,A -85,B 0,C 180,E1 -24578.69,E2 -24578.69} C_VEL
LIN {X 0,Y 140.844,Z 477.243,A -85,B 0,C 180,E1 -24581.094,E2 -24581.094} C_VEL
LIN {X 0,Y 139.251,Z 477.031,A -85,B 0,C 180,E1 -24585.107,E2 -24585.107} C_VEL
LIN {X 0,Y 138.348,Z 476.259,A -85,B 0,C 180,E1 -24589.174,E2 -24589.174} C_VEL
LIN {X 0,Y 139.256,Z 475.399,A -85,B 0,C 180,E1 -24591.556,E2 -24591.556} C_VEL
LIN {X 0,Y 143.293,Z 472.882,A -85,B 0,C 180,E1 -24596.189,E2 -24596.189} C_VEL
LIN {X 0,Y 147.643,Z 469.671,A -85,B 0,C 180,E1 -24599.982,E2 -24599.982} C_VEL
LIN {X 0,Y 153.287,Z 464.701,A -85,B 0,C 180,E1 -24604.149,E2 -24604.149} C_VEL
LIN {X 0,Y 159.693,Z 458.182,A -85,B 0,C 180,E1 -24608.028,E2 -24608.028} C_VEL
LIN {X 0,Y 165.916,Z 451.132,A -85,B 0,C 180,E1 -24611.032,E2 -24611.032} C_VEL
LIN {X 0,Y 172.641,Z 442.497,A -85,B 0,C 180,E1 -24613.786,E2 -24613.786} C_VEL
LIN {X 0,Y 178.535,Z 433.74,A -85,B 0,C 180,E1 -24615.917,E2 -24615.917} C_VEL
LIN {X 0,Y 184.712,Z 423.001,A -85,B 0,C 180,E1 -24617.891,E2 -24617.891} C_VEL
LIN {X 0,Y 190.527,Z 410.831,A -85,B 0,C 180,E1 -24619.528,E2 -24619.528} C_VEL
LIN {X 0,Y 195.174,Z 398.719,A -85,B 0,C 180,E1 -24620.725,E2 -24620.725} C_VEL
LIN {X 0,Y 199.186,Z 385.133,A -85,B 0,C 180,E1 -24621.656,E2 -24621.656} C_VEL
LIN {X 0,Y 201.818,Z 372.367,A -85,B 0,C 180,E1 -24622.261,E2 -24622.261} C_VEL
LIN {X 0,Y 204.194,Z 353.454,A -85,B 0,C 180,E1 -24622.956,E2 -24622.956} C_VEL
LIN {X 0,Y 202.3,Z 347.781,A -85,B 0,C 180,E1 -24625.294,E2 -24625.294} C_VEL
LIN {X 0,Y 200.881,Z 343.958,A -85,B 0,C 180,E1 -24627.388,E2 -24627.388} C_VEL
LIN {X 0,Y 199.888,Z 341.306,A -85,B 0,C 180,E1 -24629.102,E2 -24629.102} C_VEL
LIN {X 0,Y 198.737,Z 338.208,A -85,B 0,C 180,E1 -24631.751,E2 -24631.751} C_VEL
LIN {X 0,Y 197.632,Z 335.604,A -85,B 0,C 180,E1 -24636.371,E2 -24636.371} C_VEL
LIN {X 0,Y 197.676,Z 335.479,A -85,B 0,C 180,E1 -24640.069,E2 -24640.069} C_VEL
LIN {X 0,Y 198.175,Z 336.447,A -85,B 0,C 180,E1 -24642.699,E2 -24642.699} C_VEL
LIN {X 0,Y 199.452,Z 338.39,A -85,B 0,C 180,E1 -24645.849,E2 -24645.849} C_VEL
LIN {X 0,Y 200.982,Z 341.843,A -85,B 0,C 180,E1 -24648.606,E2 -24648.606} C_VEL
LIN {X 0,Y 202.711,Z 345.552,A -85,B 0,C 180,E1 -24651.023,E2 -24651.023} C_VEL
LIN {X 0,Y 204.457,Z 350.714,A -85,B 0,C 180,E1 -24653.164,E2 -24653.164} C_VEL
LIN {X 0,Y 201.43,Z 373.669,A -85,B 0,C 180,E1 -24654.046,E2 -24654.046} C_VEL
LIN {X 0,Y 198.725,Z 385.856,A -85,B 0,C 180,E1 -24654.695,E2 -24654.695} C_VEL
LIN {X 0,Y 195.224,Z 397.422,A -85,B 0,C 180,E1 -24655.561,E2 -24655.561} C_VEL
LIN {X 0,Y 190.001,Z 410.819,A -85,B 0,C 180,E1 -24657.006,E2 -24657.006} C_VEL
LIN {X 0,Y 184.882,Z 421.468,A -85,B 0,C 180,E1 -24658.55,E2 -24658.55} C_VEL
LIN {X 0,Y 179.175,Z 431.316,A -85,B 0,C 180,E1 -24660.39,E2 -24660.39} C_VEL
LIN {X 0,Y 172.701,Z 440.873,A -85,B 0,C 180,E1 -24662.781,E2 -24662.781} C_VEL
LIN {X 0,Y 166.588,Z 448.681,A -85,B 0,C 180,E1 -24665.354,E2 -24665.354} C_VEL
LIN {X 0,Y 160.9,Z 455.102,A -85,B 0,C 180,E1 -24668.119,E2 -24668.119} C_VEL
LIN {X 0,Y 154.413,Z 461.518,A -85,B 0,C 180,E1 -24671.8,E2 -24671.8} C_VEL
LIN {X 0,Y 149.923,Z 465.451,A -85,B 0,C 180,E1 -24674.927,E2 -24674.927} C_VEL
LIN {X 0,Y 145.662,Z 468.732,A -85,B 0,C 180,E1 -24678.435,E2 -24678.435} C_VEL
LIN {X 0,Y 140.809,Z 471.876,A -85,B 0,C 180,E1 -24683.512,E2 -24683.512} C_VEL
LIN {X 0,Y 136.948,Z 473.574,A -85,B 0,C 180,E1 -24689.271,E2 -24689.271} C_VEL
LIN {X 0,Y 134.46,Z 473.725,A -85,B 0,C 180,E1 -24695.069,E2 -24695.069} C_VEL
LIN {X 0,Y 133.493,Z 472.927,A -85,B 0,C 180,E1 -24699.152,E2 -24699.152} C_VEL
LIN {X 0,Y 132.949,Z 471.375,A -85,B 0,C 180,E1 -24703.379,E2 -24703.379} C_VEL
LIN {X 0,Y 132.91,Z 468.944,A -85,B 0,C 180,E1 -24707.722,E2 -24707.722} C_VEL
LIN {X 0,Y 133.569,Z 464.222,A -85,B 0,C 180,E1 -24713.478,E2 -24713.478} C_VEL
LIN {X 0,Y 134.721,Z 458.481,A -85,B 0,C 180,E1 -24718.562,E2 -24718.562} C_VEL
LIN {X 0,Y 136.428,Z 451.554,A -85,B 0,C 180,E1 -24723.214,E2 -24723.214} C_VEL
LIN {X 0,Y 138.678,Z 443.019,A -85,B 0,C 180,E1 -24727.666,E2 -24727.666} C_VEL
LIN {X 0,Y 141.307,Z 433.596,A -85,B 0,C 180,E1 -24731.497,E2 -24731.497} C_VEL
LIN {X 0,Y 144.085,Z 423.39,A -85,B 0,C 180,E1 -24734.722,E2 -24734.722} C_VEL
LIN {X 0,Y 147,Z 411.763,A -85,B 0,C 180,E1 -24737.581,E2 -24737.581} C_VEL
LIN {X 0,Y 149.327,Z 400.763,A -85,B 0,C 180,E1 -24739.657,E2 -24739.657} C_VEL
LIN {X 0,Y 151.464,Z 388.807,A -85,B 0,C 180,E1 -24741.356,E2 -24741.356} C_VEL
LIN {X 0,Y 153.321,Z 375.109,A -85,B 0,C 180,E1 -24742.738,E2 -24742.738} C_VEL
LIN {X 0,Y 154.668,Z 360.582,A -85,B 0,C 180,E1 -24743.613,E2 -24743.613} C_VEL
LIN {X 0,Y 157.573,Z 318.514,A -85,B 0,C 180,E1 -24745.709,E2 -24745.709} C_VEL
LIN {X 0,Y 150.388,Z 297.375,A -85,B 0,C 180,E1 -24748.561,E2 -24748.561} C_VEL
LIN {X 0,Y 140.938,Z 277.736,A -85,B 0,C 180,E1 -24752.247,E2 -24752.247} C_VEL
LIN {X 0,Y 138.117,Z 273.398,A -85,B 0,C 180,E1 -24753.342,E2 -24753.342} C_VEL
LIN {X 0,Y 136.799,Z 270.849,A -85,B 0,C 180,E1 -24754.056,E2 -24754.056} C_VEL
LIN {X 0,Y 136.568,Z 270.011,A -85,B 0,C 180,E1 -24754.802,E2 -24754.802} C_VEL
LIN {X 0,Y 136.526,Z 269.962,A -85,B 0,C 180,E1 -24758.889,E2 -24758.889} C_VEL
LIN {X 0,Y 136.407,Z 269.976,A -85,B 0,C 180,E1 -24761.898,E2 -24761.898} C_VEL
LIN {X 0,Y 136.152,Z 269.993,A -85,B 0,C 180,E1 -24768.047,E2 -24768.047} C_VEL
LIN {X 0,Y 136.148,Z 270.021,A -85,B 0,C 180,E1 -24771.758,E2 -24771.758} C_VEL
LIN {X 0,Y 136.055,Z 269.989,A -85,B 0,C 180,E1 -24778.628,E2 -24778.628} C_VEL
LIN {X 0,Y 136.043,Z 270.04,A -85,B 0,C 180,E1 -24784.635,E2 -24784.635} C_VEL
LIN {X 0,Y 136.054,Z 270.023,A -85,B 0,C 180,E1 -24789.245,E2 -24789.245} C_VEL
LIN {X 0,Y 136.071,Z 270.034,A -85,B 0,C 180,E1 -24793.722,E2 -24793.722} C_VEL
LIN {X 0,Y 136.09,Z 270.019,A -85,B 0,C 180,E1 -24797.858,E2 -24797.858} C_VEL
LIN {X 0,Y 136.098,Z 270.03,A -85,B 0,C 180,E1 -24801.736,E2 -24801.736} C_VEL
LIN {X 0,Y 136.073,Z 270.016,A -85,B 0,C 180,E1 -24805.736,E2 -24805.736} C_VEL
LIN {X 0,Y 136.129,Z 270.019,A -85,B 0,C 180,E1 -24812.337,E2 -24812.337} C_VEL
LIN {X 0,Y 136.182,Z 270.02,A -85,B 0,C 180,E1 -24818.845,E2 -24818.845} C_VEL
LIN {X 0,Y 136.227,Z 269.998,A -85,B 0,C 180,E1 -24825.073,E2 -24825.073} C_VEL
LIN {X 0,Y 136.426,Z 269.99,A -85,B 0,C 180,E1 -24828.198,E2 -24828.198} C_VEL
LIN {X 0,Y 136.539,Z 269.965,A -85,B 0,C 180,E1 -24831.137,E2 -24831.137} C_VEL
LIN {X 0,Y 137.121,Z 269.893,A -85,B 0,C 180,E1 -24840.019,E2 -24840.019} C_VEL
LIN {X 0,Y 136.551,Z 269.946,A -85,B 0,C 180,E1 -24848.901,E2 -24848.901} C_VEL
LIN {X 0,Y 136.433,Z 269.989,A -85,B 0,C 180,E1 -24851.91,E2 -24851.91} C_VEL
LIN {X 0,Y 136.19,Z 269.978,A -85,B 0,C 180,E1 -24858.056,E2 -24858.056} C_VEL
LIN {X 0,Y 136.177,Z 270.002,A -85,B 0,C 180,E1 -24861.714,E2 -24861.714} C_VEL
LIN {X 0,Y 136.12,Z 269.999,A -85,B 0,C 180,E1 -24868.622,E2 -24868.622} C_VEL
LIN {X 0,Y 136.071,Z 270.021,A -85,B 0,C 180,E1 -24874.642,E2 -24874.642} C_VEL
LIN {X 0,Y 136.004,Z 270.059,A -85,B 0,C 180,E1 -24880.573,E2 -24880.573} C_VEL
LIN {X 0,Y 136.099,Z 270.572,A -85,B 0,C 180,E1 -24881.359,E2 -24881.359} C_VEL
LIN {X 0,Y 136.815,Z 272.535,A -85,B 0,C 180,E1 -24881.999,E2 -24881.999} C_VEL
LIN {X 0,Y 138.325,Z 274.978,A -85,B 0,C 180,E1 -24882.618,E2 -24882.618} C_VEL
LIN {X 0,Y 144.575,Z 286.299,A -85,B 0,C 180,E1 -24885.087,E2 -24885.087} C_VEL
LIN {X 0,Y 150.175,Z 300.125,A -85,B 0,C 180,E1 -24887.359,E2 -24887.359} C_VEL
LIN {X 0,Y 157.07,Z 320.318,A -85,B 0,C 180,E1 -24890.089,E2 -24890.089} C_VEL
LIN {X 0,Y 157.393,Z 324.474,A -85,B 0,C 180,E1 -24890.411,E2 -24890.411} C_VEL
LIN {X 0,Y 153.815,Z 374.029,A -85,B 0,C 180,E1 -24892.923,E2 -24892.923} C_VEL
LIN {X 0,Y 152.291,Z 387.245,A -85,B 0,C 180,E1 -24894.054,E2 -24894.054} C_VEL
LIN {X 0,Y 150.195,Z 399.991,A -85,B 0,C 180,E1 -24895.632,E2 -24895.632} C_VEL
LIN {X 0,Y 147.625,Z 411.732,A -85,B 0,C 180,E1 -24897.612,E2 -24897.612} C_VEL
LIN {X 0,Y 144.88,Z 423.18,A -85,B 0,C 180,E1 -24900.179,E2 -24900.179} C_VEL
LIN {X 0,Y 142.387,Z 432.757,A -85,B 0,C 180,E1 -24902.922,E2 -24902.922} C_VEL
LIN {X 0,Y 139.792,Z 442.088,A -85,B 0,C 180,E1 -24906.279,E2 -24906.279} C_VEL
LIN {X 0,Y 137.268,Z 451.316,A -85,B 0,C 180,E1 -24910.557,E2 -24910.557} C_VEL
LIN {X 0,Y 135.365,Z 458.724,A -85,B 0,C 180,E1 -24914.949,E2 -24914.949} C_VEL
LIN {X 0,Y 134.216,Z 464.636,A -85,B 0,C 180,E1 -24919.435,E2 -24919.435} C_VEL
LIN {X 0,Y 133.578,Z 469.236,A -85,B 0,C 180,E1 -24923.955,E2 -24923.955} C_VEL
LIN {X 0,Y 133.437,Z 471.638,A -85,B 0,C 180,E1 -24926.976,E2 -24926.976} C_VEL
LIN {X 0,Y 133.531,Z 473.593,A -85,B 0,C 180,E1 -24929.995,E2 -24929.995} C_VEL
LIN {X 0,Y 133.433,Z 475.1,A -85,B 0,C 180,E1 -24933.014,E2 -24933.014} C_VEL
LIN {X 0,Y 133.545,Z 476.168,A -85,B 0,C 180,E1 -24936.036,E2 -24936.036} C_VEL
LIN {X 0,Y 134.674,Z 477.122,A -85,B 0,C 180,E1 -24942.043,E2 -24942.043} C_VEL
LIN {X 0,Y 137.033,Z 476.599,A -85,B 0,C 180,E1 -24947.916,E2 -24947.916} C_VEL
LIN {X 0,Y 139.256,Z 475.399,A -85,B 0,C 180,E1 -24951.556,E2 -24951.556} C_VEL
LIN {X 0,Y 140.434,Z 474.404,A -85,B 0,C 180,E1 -24953.892,E2 -24953.892} C_VEL
LIN {X 0,Y 141.161,Z 472.382,A -85,B 0,C 180,E1 -24957.843,E2 -24957.843} C_VEL
LIN {X 0,Y 142.549,Z 469.812,A -85,B 0,C 180,E1 -24961.665,E2 -24961.665} C_VEL
LIN {X 0,Y 144.68,Z 467.823,A -85,B 0,C 180,E1 -24963.713,E2 -24963.713} C_VEL
LIN {X 0,Y 150.309,Z 462.938,A -85,B 0,C 180,E1 -24967.427,E2 -24967.427} C_VEL
LIN {X 0,Y 157.338,Z 456.029,A -85,B 0,C 180,E1 -24971.206,E2 -24971.206} C_VEL
LIN {X 0,Y 164.119,Z 448.558,A -85,B 0,C 180,E1 -24974.09,E2 -24974.09} C_VEL
LIN {X 0,Y 171.34,Z 439.274,A -85,B 0,C 180,E1 -24976.718,E2 -24976.718} C_VEL
LIN {X 0,Y 178.226,Z 428.847,A -85,B 0,C 180,E1 -24978.945,E2 -24978.945} C_VEL
LIN {X 0,Y 184.166,Z 418.246,A -85,B 0,C 180,E1 -24980.596,E2 -24980.596} C_VEL
LIN {X 0,Y 189.537,Z 406.516,A -85,B 0,C 180,E1 -24981.987,E2 -24981.987} C_VEL
LIN {X 0,Y 194.072,Z 394.249,A -85,B 0,C 180,E1 -24983.016,E2 -24983.016} C_VEL
LIN {X 0,Y 197.569,Z 381.509,A -85,B 0,C 180,E1 -24983.767,E2 -24983.767} C_VEL
LIN {X 0,Y 200.164,Z 367.139,A -85,B 0,C 180,E1 -24984.363,E2 -24984.363} C_VEL
LIN {X 0,Y 201.38,Z 357.068,A -85,B 0,C 180,E1 -24984.751,E2 -24984.751} C_VEL
LIN {X 0,Y 199.772,Z 351.857,A -85,B 0,C 180,E1 -24987.187,E2 -24987.187} C_VEL
LIN {X 0,Y 198.324,Z 347.774,A -85,B 0,C 180,E1 -24989.804,E2 -24989.804} C_VEL
LIN {X 0,Y 197.337,Z 344.908,A -85,B 0,C 180,E1 -24992.407,E2 -24992.407} C_VEL
LIN {X 0,Y 196.474,Z 342.504,A -85,B 0,C 180,E1 -24996.816,E2 -24996.816} C_VEL
LIN {X 0,Y 196.682,Z 342.646,A -85,B 0,C 180,E1 -25000.868,E2 -25000.868} C_VEL
LIN {X 0,Y 198.089,Z 345.198,A -85,B 0,C 180,E1 -25005.393,E2 -25005.393} C_VEL
LIN {X 0,Y 199.654,Z 349.045,A -85,B 0,C 180,E1 -25008.429,E2 -25008.429} C_VEL
LIN {X 0,Y 200.826,Z 351.828,A -85,B 0,C 180,E1 -25010.202,E2 -25010.202} C_VEL
LIN {X 0,Y 201.679,Z 354.579,A -85,B 0,C 180,E1 -25011.428,E2 -25011.428} C_VEL
LIN {X 0,Y 198.843,Z 374.581,A -85,B 0,C 180,E1 -25012.169,E2 -25012.169} C_VEL
LIN {X 0,Y 195.891,Z 387.156,A -85,B 0,C 180,E1 -25012.832,E2 -25012.832} C_VEL
LIN {X 0,Y 192.243,Z 398.516,A -85,B 0,C 180,E1 -25013.69,E2 -25013.69} C_VEL
LIN {X 0,Y 187.384,Z 410.436,A -85,B 0,C 180,E1 -25014.939,E2 -25014.939} C_VEL
LIN {X 0,Y 181.621,Z 421.922,A -85,B 0,C 180,E1 -25016.57,E2 -25016.57} C_VEL
LIN {X 0,Y 175.014,Z 432.623,A -85,B 0,C 180,E1 -25018.582,E2 -25018.582} C_VEL
LIN {X 0,Y 168.017,Z 442.357,A -85,B 0,C 180,E1 -25021.06,E2 -25021.06} C_VEL
LIN {X 0,Y 161.934,Z 449.624,A -85,B 0,C 180,E1 -25023.515,E2 -25023.515} C_VEL
LIN {X 0,Y 155.593,Z 456.251,A -85,B 0,C 180,E1 -25026.472,E2 -25026.472} C_VEL
LIN {X 0,Y 149.691,Z 461.606,A -85,B 0,C 180,E1 -25029.648,E2 -25029.648} C_VEL
LIN {X 0,Y 142.933,Z 466.961,A -85,B 0,C 180,E1 -25034.212,E2 -25034.212} C_VEL
LIN {X 0,Y 138.782,Z 469.783,A -85,B 0,C 180,E1 -25037.667,E2 -25037.667} C_VEL
LIN {X 0,Y 135.168,Z 471.849,A -85,B 0,C 180,E1 -25041.321,E2 -25041.321} C_VEL
LIN {X 0,Y 132.086,Z 473.211,A -85,B 0,C 180,E1 -25045.254,E2 -25045.254} C_VEL
LIN {X 0,Y 129.451,Z 473.904,A -85,B 0,C 180,E1 -25049.71,E2 -25049.71} C_VEL
LIN {X 0,Y 127.548,Z 473.775,A -85,B 0,C 180,E1 -25054.269,E2 -25054.269} C_VEL
LIN {X 0,Y 126.416,Z 472.797,A -85,B 0,C 180,E1 -25058.903,E2 -25058.903} C_VEL
LIN {X 0,Y 125.843,Z 471.018,A -85,B 0,C 180,E1 -25063.456,E2 -25063.456} C_VEL
LIN {X 0,Y 125.825,Z 468.475,A -85,B 0,C 180,E1 -25067.921,E2 -25067.921} C_VEL
LIN {X 0,Y 126.229,Z 465.181,A -85,B 0,C 180,E1 -25072.241,E2 -25072.241} C_VEL
LIN {X 0,Y 127.311,Z 459.91,A -85,B 0,C 180,E1 -25077.443,E2 -25077.443} C_VEL
LIN {X 0,Y 129.007,Z 452.849,A -85,B 0,C 180,E1 -25082.722,E2 -25082.722} C_VEL
LIN {X 0,Y 131.049,Z 445.272,A -85,B 0,C 180,E1 -25087.098,E2 -25087.098} C_VEL
LIN {X 0,Y 133.63,Z 436.36,A -85,B 0,C 180,E1 -25091.132,E2 -25091.132} C_VEL
LIN {X 0,Y 136.45,Z 426.341,A -85,B 0,C 180,E1 -25094.7,E2 -25094.7} C_VEL
LIN {X 0,Y 139.348,Z 415.714,A -85,B 0,C 180,E1 -25097.628,E2 -25097.628} C_VEL
LIN {X 0,Y 142.052,Z 404.078,A -85,B 0,C 180,E1 -25100.104,E2 -25100.104} C_VEL
LIN {X 0,Y 144.566,Z 391.264,A -85,B 0,C 180,E1 -25102.146,E2 -25102.146} C_VEL
LIN {X 0,Y 146.588,Z 377.386,A -85,B 0,C 180,E1 -25103.683,E2 -25103.683} C_VEL
LIN {X 0,Y 148.005,Z 364.232,A -85,B 0,C 180,E1 -25104.596,E2 -25104.596} C_VEL
LIN {X 0,Y 151.127,Z 319.578,A -85,B 0,C 180,E1 -25106.917,E2 -25106.917} C_VEL
LIN {X 0,Y 144.539,Z 300.183,A -85,B 0,C 180,E1 -25109.729,E2 -25109.729} C_VEL
LIN {X 0,Y 135.814,Z 281.975,A -85,B 0,C 180,E1 -25113.335,E2 -25113.335} C_VEL
LIN {X 0,Y 131.153,Z 274.564,A -85,B 0,C 180,E1 -25115.334,E2 -25115.334} C_VEL
LIN {X 0,Y 129.754,Z 272.185,A -85,B 0,C 180,E1 -25116.03,E2 -25116.03} C_VEL
LIN {X 0,Y 129.456,Z 270.954,A -85,B 0,C 180,E1 -25116.826,E2 -25116.826} C_VEL
LIN {X 0,Y 129.35,Z 270.857,A -85,B 0,C 180,E1 -25122.157,E2 -25122.157} C_VEL
LIN {X 0,Y 129.076,Z 270.875,A -85,B 0,C 180,E1 -25129.073,E2 -25129.073} C_VEL
LIN {X 0,Y 129.062,Z 270.907,A -85,B 0,C 180,E1 -25132.412,E2 -25132.412} C_VEL
LIN {X 0,Y 128.975,Z 270.87,A -85,B 0,C 180,E1 -25139.374,E2 -25139.374} C_VEL
LIN {X 0,Y 128.986,Z 270.918,A -85,B 0,C 180,E1 -25145.226,E2 -25145.226} C_VEL
LIN {X 0,Y 128.982,Z 270.912,A -85,B 0,C 180,E1 -25150.84,E2 -25150.84} C_VEL
LIN {X 0,Y 129.001,Z 270.905,A -85,B 0,C 180,E1 -25155.099,E2 -25155.099} C_VEL
LIN {X 0,Y 129.025,Z 270.91,A -85,B 0,C 180,E1 -25159.699,E2 -25159.699} C_VEL
LIN {X 0,Y 129.008,Z 270.896,A -85,B 0,C 180,E1 -25164.809,E2 -25164.809} C_VEL
LIN {X 0,Y 129.001,Z 270.916,A -85,B 0,C 180,E1 -25170.664,E2 -25170.664} C_VEL
LIN {X 0,Y 129.064,Z 270.903,A -85,B 0,C 180,E1 -25177.617,E2 -25177.617} C_VEL
LIN {X 0,Y 129.147,Z 270.876,A -85,B 0,C 180,E1 -25184.234,E2 -25184.234} C_VEL
LIN {X 0,Y 129.344,Z 270.873,A -85,B 0,C 180,E1 -25187.992,E2 -25187.992} C_VEL
LIN {X 0,Y 129.464,Z 270.85,A -85,B 0,C 180,E1 -25190.649,E2 -25190.649} C_VEL
LIN {X 0,Y 130.076,Z 270.77,A -85,B 0,C 180,E1 -25200.02,E2 -25200.02} C_VEL
LIN {X 0,Y 129.478,Z 270.832,A -85,B 0,C 180,E1 -25209.392,E2 -25209.392} C_VEL
LIN {X 0,Y 129.317,Z 270.878,A -85,B 0,C 180,E1 -25212.576,E2 -25212.576} C_VEL
LIN {X 0,Y 129.108,Z 270.858,A -85,B 0,C 180,E1 -25219.084,E2 -25219.084} C_VEL
LIN {X 0,Y 129.098,Z 270.892,A -85,B 0,C 180,E1 -25222.421,E2 -25222.421} C_VEL
LIN {X 0,Y 129.046,Z 270.88,A -85,B 0,C 180,E1 -25229.372,E2 -25229.372} C_VEL
LIN {X 0,Y 128.986,Z 270.898,A -85,B 0,C 180,E1 -25235.177,E2 -25235.177} C_VEL
LIN {X 0,Y 129.053,Z 271.049,A -85,B 0,C 180,E1 -25238.946,E2 -25238.946} C_VEL
LIN {X 0,Y 129.265,Z 272.191,A -85,B 0,C 180,E1 -25239.609,E2 -25239.609} C_VEL
LIN {X 0,Y 130.901,Z 274.989,A -85,B 0,C 180,E1 -25240.386,E2 -25240.386} C_VEL
LIN {X 0,Y 139.103,Z 289.87,A -85,B 0,C 180,E1 -25243.949,E2 -25243.949} C_VEL
LIN {X 0,Y 144.462,Z 303.22,A -85,B 0,C 180,E1 -25246.254,E2 -25246.254} C_VEL
LIN {X 0,Y 150.834,Z 322.094,A -85,B 0,C 180,E1 -25248.97,E2 -25248.97} C_VEL
LIN {X 0,Y 151.109,Z 324.787,A -85,B 0,C 180,E1 -25249.204,E2 -25249.204} C_VEL
LIN {X 0,Y 147.375,Z 374.123,A -85,B 0,C 180,E1 -25251.792,E2 -25251.792} C_VEL
LIN {X 0,Y 145.689,Z 387.845,A -85,B 0,C 180,E1 -25253.018,E2 -25253.018} C_VEL
LIN {X 0,Y 143.537,Z 400.412,A -85,B 0,C 180,E1 -25254.659,E2 -25254.659} C_VEL
LIN {X 0,Y 140.891,Z 412.024,A -85,B 0,C 180,E1 -25256.716,E2 -25256.716} C_VEL
LIN {X 0,Y 138.039,Z 423.4,A -85,B 0,C 180,E1 -25259.389,E2 -25259.389} C_VEL
LIN {X 0,Y 135.228,Z 433.739,A -85,B 0,C 180,E1 -25262.527,E2 -25262.527} C_VEL
LIN {X 0,Y 132.292,Z 443.856,A -85,B 0,C 180,E1 -25266.514,E2 -25266.514} C_VEL
LIN {X 0,Y 130.171,Z 451.39,A -85,B 0,C 180,E1 -25270.274,E2 -25270.274} C_VEL
LIN {X 0,Y 128.237,Z 458.77,A -85,B 0,C 180,E1 -25274.905,E2 -25274.905} C_VEL
LIN {X 0,Y 127.219,Z 463.738,A -85,B 0,C 180,E1 -25278.846,E2 -25278.846} C_VEL
LIN {X 0,Y 126.536,Z 468.521,A -85,B 0,C 180,E1 -25283.617,E2 -25283.617} C_VEL
LIN {X 0,Y 126.35,Z 472.118,A -85,B 0,C 180,E1 -25288.401,E2 -25288.401} C_VEL
LIN {X 0,Y 126.456,Z 473.083,A -85,B 0,C 180,E1 -25289.995,E2 -25289.995} C_VEL
LIN {X 0,Y 126.376,Z 474.657,A -85,B 0,C 180,E1 -25293.182,E2 -25293.182} C_VEL
LIN {X 0,Y 126.937,Z 476.612,A -85,B 0,C 180,E1 -25299.555,E2 -25299.555} C_VEL
LIN {X 0,Y 128.81,Z 476.982,A -85,B 0,C 180,E1 -25305.825,E2 -25305.825} C_VEL
LIN {X 0,Y 132.061,Z 475.889,A -85,B 0,C 180,E1 -25311.865,E2 -25311.865} C_VEL
LIN {X 0,Y 134.337,Z 474.777,A -85,B 0,C 180,E1 -25314.736,E2 -25314.736} C_VEL
LIN {X 0,Y 139.952,Z 471.318,A -85,B 0,C 180,E1 -25320.138,E2 -25320.138} C_VEL
LIN {X 0,Y 144.68,Z 467.823,A -85,B 0,C 180,E1 -25323.713,E2 -25323.713} C_VEL
LIN {X 0,Y 146.932,Z 465.71,A -85,B 0,C 180,E1 -25325.694,E2 -25325.694} C_VEL
LIN {X 0,Y 149.249,Z 462.115,A -85,B 0,C 180,E1 -25329.167,E2 -25329.167} C_VEL
LIN {X 0,Y 151.93,Z 457.886,A -85,B 0,C 180,E1 -25332.413,E2 -25332.413} C_VEL
LIN {X 0,Y 154.621,Z 454.787,A -85,B 0,C 180,E1 -25333.984,E2 -25333.984} C_VEL
LIN {X 0,Y 161.627,Z 447.234,A -85,B 0,C 180,E1 -25336.74,E2 -25336.74} C_VEL
LIN {X 0,Y 169.222,Z 437.784,A -85,B 0,C 180,E1 -25339.276,E2 -25339.276} C_VEL
LIN {X 0,Y 175.799,Z 428.116,A -85,B 0,C 180,E1 -25341.213,E2 -25341.213} C_VEL
LIN {X 0,Y 181.956,Z 417.335,A -85,B 0,C 180,E1 -25342.803,E2 -25342.803} C_VEL
LIN {X 0,Y 187.521,Z 405.404,A -85,B 0,C 180,E1 -25344.135,E2 -25344.135} C_VEL
LIN {X 0,Y 192.19,Z 392.774,A -85,B 0,C 180,E1 -25345.118,E2 -25345.118} C_VEL
LIN {X 0,Y 195.845,Z 379.473,A -85,B 0,C 180,E1 -25345.83,E2 -25345.83} C_VEL
LIN {X 0,Y 198.27,Z 365.597,A -85,B 0,C 180,E1 -25346.381,E2 -25346.381} C_VEL
LIN {X 0,Y 198.845,Z 360.997,A -85,B 0,C 180,E1 -25346.57,E2 -25346.57} C_VEL
LIN {X 0,Y 197.654,Z 357.006,A -85,B 0,C 180,E1 -25348.699,E2 -25348.699} C_VEL
LIN {X 0,Y 196.789,Z 354.147,A -85,B 0,C 180,E1 -25350.636,E2 -25350.636} C_VEL
LIN {X 0,Y 196.031,Z 351.732,A -85,B 0,C 180,E1 -25352.874,E2 -25352.874} C_VEL
LIN {X 0,Y 195.368,Z 349.566,A -85,B 0,C 180,E1 -25356.677,E2 -25356.677} C_VEL
LIN {X 0,Y 195.545,Z 349.644,A -85,B 0,C 180,E1 -25360.752,E2 -25360.752} C_VEL
LIN {X 0,Y 196.731,Z 351.979,A -85,B 0,C 180,E1 -25364.91,E2 -25364.91} C_VEL
LIN {X 0,Y 197.994,Z 355.465,A -85,B 0,C 180,E1 -25367.69,E2 -25367.69} C_VEL
LIN {X 0,Y 198.983,Z 357.958,A -85,B 0,C 180,E1 -25369.316,E2 -25369.316} C_VEL
LIN {X 0,Y 199.143,Z 358.616,A -85,B 0,C 180,E1 -25369.605,E2 -25369.605} C_VEL
LIN {X 0,Y 196.446,Z 376.013,A -85,B 0,C 180,E1 -25370.26,E2 -25370.26} C_VEL
LIN {X 0,Y 193.361,Z 388.158,A -85,B 0,C 180,E1 -25370.898,E2 -25370.898} C_VEL
LIN {X 0,Y 189.131,Z 400.462,A -85,B 0,C 180,E1 -25371.834,E2 -25371.834} C_VEL
LIN {X 0,Y 184.054,Z 412.22,A -85,B 0,C 180,E1 -25373.079,E2 -25373.079} C_VEL
LIN {X 0,Y 178.133,Z 423.249,A -85,B 0,C 180,E1 -25374.647,E2 -25374.647} C_VEL
LIN {X 0,Y 171.269,Z 433.801,A -85,B 0,C 180,E1 -25376.636,E2 -25376.636} C_VEL
LIN {X 0,Y 164.092,Z 443.14,A -85,B 0,C 180,E1 -25379.031,E2 -25379.031} C_VEL
LIN {X 0,Y 156.599,Z 451.376,A -85,B 0,C 180,E1 -25381.912,E2 -25381.912} C_VEL
LIN {X 0,Y 149.019,Z 458.59,A -85,B 0,C 180,E1 -25385.394,E2 -25385.394} C_VEL
LIN {X 0,Y 142.326,Z 464.01,A -85,B 0,C 180,E1 -25389.072,E2 -25389.072} C_VEL
LIN {X 0,Y 136.886,Z 467.806,A -85,B 0,C 180,E1 -25392.736,E2 -25392.736} C_VEL
LIN {X 0,Y 132.065,Z 470.653,A -85,B 0,C 180,E1 -25396.707,E2 -25396.707} C_VEL
LIN {X 0,Y 127.921,Z 472.629,A -85,B 0,C 180,E1 -25400.953,E2 -25400.953} C_VEL
LIN {X 0,Y 123.586,Z 473.97,A -85,B 0,C 180,E1 -25407.035,E2 -25407.035} C_VEL
LIN {X 0,Y 121.456,Z 473.991,A -85,B 0,C 180,E1 -25411.357,E2 -25411.357} C_VEL
LIN {X 0,Y 119.938,Z 473.353,A -85,B 0,C 180,E1 -25415.841,E2 -25415.841} C_VEL
LIN {X 0,Y 119.048,Z 471.98,A -85,B 0,C 180,E1 -25420.462,E2 -25420.462} C_VEL
LIN {X 0,Y 118.679,Z 469.739,A -85,B 0,C 180,E1 -25425.25,E2 -25425.25} C_VEL
LIN {X 0,Y 118.896,Z 466.546,A -85,B 0,C 180,E1 -25430.174,E2 -25430.174} C_VEL
LIN {X 0,Y 119.686,Z 462.162,A -85,B 0,C 180,E1 -25435.25,E2 -25435.25} C_VEL
LIN {X 0,Y 121.038,Z 456.222,A -85,B 0,C 180,E1 -25440.52,E2 -25440.52} C_VEL
LIN {X 0,Y 122.885,Z 449.436,A -85,B 0,C 180,E1 -25445.216,E2 -25445.216} C_VEL
LIN {X 0,Y 125.447,Z 440.65,A -85,B 0,C 180,E1 -25449.938,E2 -25449.938} C_VEL
LIN {X 0,Y 128.445,Z 430.597,A -85,B 0,C 180,E1 -25454.128,E2 -25454.128} C_VEL
LIN {X 0,Y 131.334,Z 420.724,A -85,B 0,C 180,E1 -25457.311,E2 -25457.311} C_VEL
LIN {X 0,Y 134.339,Z 409.033,A -85,B 0,C 180,E1 -25460.218,E2 -25460.218} C_VEL
LIN {X 0,Y 137.006,Z 397.153,A -85,B 0,C 180,E1 -25462.452,E2 -25462.452} C_VEL
LIN {X 0,Y 139.326,Z 383.884,A -85,B 0,C 180,E1 -25464.256,E2 -25464.256} C_VEL
LIN {X 0,Y 141.063,Z 370.745,A -85,B 0,C 180,E1 -25465.457,E2 -25465.457} C_VEL
LIN {X 0,Y 144.82,Z 320.905,A -85,B 0,C 180,E1 -25468.2,E2 -25468.2} C_VEL
LIN {X 0,Y 138.708,Z 302.944,A -85,B 0,C 180,E1 -25470.966,E2 -25470.966} C_VEL
LIN {X 0,Y 130.874,Z 286.421,A -85,B 0,C 180,E1 -25474.447,E2 -25474.447} C_VEL
LIN {X 0,Y 123.889,Z 275.272,A -85,B 0,C 180,E1 -25477.683,E2 -25477.683} C_VEL
LIN {X 0,Y 122.55,Z 272.562,A -85,B 0,C 180,E1 -25478.56,E2 -25478.56} C_VEL
LIN {X 0,Y 122.421,Z 271.785,A -85,B 0,C 180,E1 -25479.297,E2 -25479.297} C_VEL
LIN {X 0,Y 122.189,Z 271.76,A -85,B 0,C 180,E1 -25483.307,E2 -25483.307} C_VEL
LIN {X 0,Y 121.979,Z 271.765,A -85,B 0,C 180,E1 -25490.23,E2 -25490.23} C_VEL
LIN {X 0,Y 121.934,Z 271.794,A -85,B 0,C 180,E1 -25493.801,E2 -25493.801} C_VEL
LIN {X 0,Y 121.888,Z 271.755,A -85,B 0,C 180,E1 -25500.18,E2 -25500.18} C_VEL
LIN {X 0,Y 121.9,Z 271.798,A -85,B 0,C 180,E1 -25506.224,E2 -25506.224} C_VEL
LIN {X 0,Y 121.911,Z 271.797,A -85,B 0,C 180,E1 -25511.496,E2 -25511.496} C_VEL
LIN {X 0,Y 121.942,Z 271.784,A -85,B 0,C 180,E1 -25518.532,E2 -25518.532} C_VEL
LIN {X 0,Y 121.959,Z 271.773,A -85,B 0,C 180,E1 -25524.842,E2 -25524.842} C_VEL
LIN {X 0,Y 121.913,Z 271.799,A -85,B 0,C 180,E1 -25529.86,E2 -25529.86} C_VEL
LIN {X 0,Y 121.947,Z 271.779,A -85,B 0,C 180,E1 -25536.233,E2 -25536.233} C_VEL
LIN {X 0,Y 121.984,Z 271.789,A -85,B 0,C 180,E1 -25539.801,E2 -25539.801} C_VEL
LIN {X 0,Y 122.187,Z 271.758,A -85,B 0,C 180,E1 -25546.722,E2 -25546.722} C_VEL
LIN {X 0,Y 122.392,Z 271.734,A -85,B 0,C 180,E1 -25550.103,E2 -25550.103} C_VEL
LIN {X 0,Y 122.57,Z 271.717,A -85,B 0,C 180,E1 -25556.735,E2 -25556.735} C_VEL
LIN {X 0,Y 123.029,Z 271.646,A -85,B 0,C 180,E1 -25560.022,E2 -25560.022} C_VEL
LIN {X 0,Y 122.416,Z 271.672,A -85,B 0,C 180,E1 -25566.615,E2 -25566.615} C_VEL
LIN {X 0,Y 122.407,Z 271.718,A -85,B 0,C 180,E1 -25569.94,E2 -25569.94} C_VEL
LIN {X 0,Y 122.207,Z 271.762,A -85,B 0,C 180,E1 -25573.32,E2 -25573.32} C_VEL
LIN {X 0,Y 122.013,Z 271.745,A -85,B 0,C 180,E1 -25580.24,E2 -25580.24} C_VEL
LIN {X 0,Y 121.988,Z 271.79,A -85,B 0,C 180,E1 -25583.806,E2 -25583.806} C_VEL
LIN {X 0,Y 121.956,Z 271.765,A -85,B 0,C 180,E1 -25590.175,E2 -25590.175} C_VEL
LIN {X 0,Y 121.959,Z 271.981,A -85,B 0,C 180,E1 -25596.539,E2 -25596.539} C_VEL
LIN {X 0,Y 122.285,Z 273.317,A -85,B 0,C 180,E1 -25597.314,E2 -25597.314} C_VEL
LIN {X 0,Y 124.777,Z 277.531,A -85,B 0,C 180,E1 -25598.615,E2 -25598.615} C_VEL
LIN {X 0,Y 130.996,Z 288.409,A -85,B 0,C 180,E1 -25601.527,E2 -25601.527} C_VEL
LIN {X 0,Y 134.864,Z 296.041,A -85,B 0,C 180,E1 -25603.261,E2 -25603.261} C_VEL
LIN {X 0,Y 140.165,Z 310.382,A -85,B 0,C 180,E1 -25605.724,E2 -25605.724} C_VEL
LIN {X 0,Y 144.811,Z 324.578,A -85,B 0,C 180,E1 -25607.837,E2 -25607.837} C_VEL
LIN {X 0,Y 141.139,Z 372.936,A -85,B 0,C 180,E1 -25610.468,E2 -25610.468} C_VEL
LIN {X 0,Y 139.5,Z 386.323,A -85,B 0,C 180,E1 -25611.656,E2 -25611.656} C_VEL
LIN {X 0,Y 137.124,Z 399.774,A -85,B 0,C 180,E1 -25613.424,E2 -25613.424} C_VEL
LIN {X 0,Y 134.185,Z 412.311,A -85,B 0,C 180,E1 -25615.728,E2 -25615.728} C_VEL
LIN {X 0,Y 131.221,Z 423.621,A -85,B 0,C 180,E1 -25618.516,E2 -25618.516} C_VEL
LIN {X 0,Y 128.319,Z 433.892,A -85,B 0,C 180,E1 -25621.805,E2 -25621.805} C_VEL
LIN {X 0,Y 125.27,Z 443.938,A -85,B 0,C 180,E1 -25625.994,E2 -25625.994} C_VEL
LIN {X 0,Y 123.055,Z 451.419,A -85,B 0,C 180,E1 -25629.954,E2 -25629.954} C_VEL
LIN {X 0,Y 121.114,Z 458.762,A -85,B 0,C 180,E1 -25634.857,E2 -25634.857} C_VEL
LIN {X 0,Y 119.93,Z 464.593,A -85,B 0,C 180,E1 -25639.869,E2 -25639.869} C_VEL
LIN {X 0,Y 119.382,Z 469.137,A -85,B 0,C 180,E1 -25644.928,E2 -25644.928} C_VEL
LIN {X 0,Y 119.368,Z 472.549,A -85,B 0,C 180,E1 -25649.994,E2 -25649.994} C_VEL
LIN {X 0,Y 119.298,Z 474.206,A -85,B 0,C 180,E1 -25653.371,E2 -25653.371} C_VEL
LIN {X 0,Y 119.949,Z 476.333,A -85,B 0,C 180,E1 -25660.118,E2 -25660.118} C_VEL
LIN {X 0,Y 120.797,Z 476.827,A -85,B 0,C 180,E1 -25663.451,E2 -25663.451} C_VEL
LIN {X 0,Y 123.535,Z 476.641,A -85,B 0,C 180,E1 -25669.953,E2 -25669.953} C_VEL
LIN {X 0,Y 127.921,Z 474.986,A -85,B 0,C 180,E1 -25676.067,E2 -25676.067} C_VEL
LIN {X 0,Y 130.742,Z 473.595,A -85,B 0,C 180,E1 -25678.927,E2 -25678.927} C_VEL
LIN {X 0,Y 137.26,Z 469.553,A -85,B 0,C 180,E1 -25684.272,E2 -25684.272} C_VEL
LIN {X 0,Y 143.489,Z 464.867,A -85,B 0,C 180,E1 -25688.377,E2 -25688.377} C_VEL
LIN {X 0,Y 151.05,Z 458.24,A -85,B 0,C 180,E1 -25692.42,E2 -25692.42} C_VEL
LIN {X 0,Y 154.621,Z 454.787,A -85,B 0,C 180,E1 -25693.984,E2 -25693.984} C_VEL
LIN {X 0,Y 157.447,Z 451.55,A -85,B 0,C 180,E1 -25695.459,E2 -25695.459} C_VEL
LIN {X 0,Y 160.959,Z 446.187,A -85,B 0,C 180,E1 -25698.188,E2 -25698.188} C_VEL
LIN {X 0,Y 164.566,Z 440.411,A -85,B 0,C 180,E1 -25700.718,E2 -25700.718} C_VEL
LIN {X 0,Y 167.383,Z 436.409,A -85,B 0,C 180,E1 -25701.858,E2 -25701.858} C_VEL
LIN {X 0,Y 174.341,Z 426.281,A -85,B 0,C 180,E1 -25703.722,E2 -25703.722} C_VEL
LIN {X 0,Y 180.737,Z 415.229,A -85,B 0,C 180,E1 -25705.222,E2 -25705.222} C_VEL
LIN {X 0,Y 185.797,Z 404.554,A -85,B 0,C 180,E1 -25706.315,E2 -25706.315} C_VEL
LIN {X 0,Y 190.631,Z 391.615,A -85,B 0,C 180,E1 -25707.241,E2 -25707.241} C_VEL
LIN {X 0,Y 194.343,Z 378.056,A -85,B 0,C 180,E1 -25707.918,E2 -25707.918} C_VEL
LIN {X 0,Y 196.526,Z 365.484,A -85,B 0,C 180,E1 -25708.39,E2 -25708.39} C_VEL
LIN {X 0,Y 195.983,Z 363.222,A -85,B 0,C 180,E1 -25709.571,E2 -25709.571} C_VEL
LIN {X 0,Y 195.281,Z 360.438,A -85,B 0,C 180,E1 -25711.538,E2 -25711.538} C_VEL
LIN {X 0,Y 194.708,Z 358.468,A -85,B 0,C 180,E1 -25713.453,E2 -25713.453} C_VEL
LIN {X 0,Y 194.257,Z 356.67,A -85,B 0,C 180,E1 -25716.536,E2 -25716.536} C_VEL
LIN {X 0,Y 194.332,Z 356.517,A -85,B 0,C 180,E1 -25720.087,E2 -25720.087} C_VEL
LIN {X 0,Y 195.265,Z 358.403,A -85,B 0,C 180,E1 -25724.06,E2 -25724.06} C_VEL
LIN {X 0,Y 196.325,Z 361.751,A -85,B 0,C 180,E1 -25726.854,E2 -25726.854} C_VEL
LIN {X 0,Y 196.826,Z 363.047,A -85,B 0,C 180,E1 -25727.772,E2 -25727.772} C_VEL
LIN {X 0,Y 194.332,Z 377.417,A -85,B 0,C 180,E1 -25728.294,E2 -25728.294} C_VEL
LIN {X 0,Y 190.919,Z 389.974,A -85,B 0,C 180,E1 -25728.959,E2 -25728.959} C_VEL
LIN {X 0,Y 186.43,Z 402.277,A -85,B 0,C 180,E1 -25729.889,E2 -25729.889} C_VEL
LIN {X 0,Y 181.273,Z 413.41,A -85,B 0,C 180,E1 -25731.064,E2 -25731.064} C_VEL
LIN {X 0,Y 174.665,Z 424.909,A -85,B 0,C 180,E1 -25732.696,E2 -25732.696} C_VEL
LIN {X 0,Y 168.113,Z 434.448,A -85,B 0,C 180,E1 -25734.489,E2 -25734.489} C_VEL
LIN {X 0,Y 160.71,Z 443.609,A -85,B 0,C 180,E1 -25736.804,E2 -25736.804} C_VEL
LIN {X 0,Y 153.598,Z 451.096,A -85,B 0,C 180,E1 -25739.356,E2 -25739.356} C_VEL
LIN {X 0,Y 145.525,Z 458.344,A -85,B 0,C 180,E1 -25742.75,E2 -25742.75} C_VEL
LIN {X 0,Y 139.444,Z 463.019,A -85,B 0,C 180,E1 -25745.766,E2 -25745.766} C_VEL
LIN {X 0,Y 133.984,Z 466.752,A -85,B 0,C 180,E1 -25749.033,E2 -25749.033} C_VEL
LIN {X 0,Y 126.759,Z 470.833,A -85,B 0,C 180,E1 -25754.425,E2 -25754.425} C_VEL
LIN {X 0,Y 120.365,Z 473.389,A -85,B 0,C 180,E1 -25760.914,E2 -25760.914} C_VEL
LIN {X 0,Y 116.992,Z 474.119,A -85,B 0,C 180,E1 -25765.714,E2 -25765.714} C_VEL
LIN {X 0,Y 114.467,Z 474.025,A -85,B 0,C 180,E1 -25770.745,E2 -25770.745} C_VEL
LIN {X 0,Y 112.783,Z 473.078,A -85,B 0,C 180,E1 -25775.907,E2 -25775.907} C_VEL
LIN {X 0,Y 111.85,Z 471.339,A -85,B 0,C 180,E1 -25781.072,E2 -25781.072} C_VEL
LIN {X 0,Y 111.59,Z 468.831,A -85,B 0,C 180,E1 -25786.158,E2 -25786.158} C_VEL
LIN {X 0,Y 111.907,Z 465.547,A -85,B 0,C 180,E1 -25791.104,E2 -25791.104} C_VEL
LIN {X 0,Y 112.937,Z 460.348,A -85,B 0,C 180,E1 -25796.95,E2 -25796.95} C_VEL
LIN {X 0,Y 114.553,Z 453.734,A -85,B 0,C 180,E1 -25802.611,E2 -25802.611} C_VEL
LIN {X 0,Y 116.394,Z 447.381,A -85,B 0,C 180,E1 -25806.898,E2 -25806.898} C_VEL
LIN {X 0,Y 119.084,Z 438.818,A -85,B 0,C 180,E1 -25811.502,E2 -25811.502} C_VEL
LIN {X 0,Y 121.88,Z 429.726,A -85,B 0,C 180,E1 -25815.331,E2 -25815.331} C_VEL
LIN {X 0,Y 124.905,Z 419.618,A -85,B 0,C 180,E1 -25818.648,E2 -25818.648} C_VEL
LIN {X 0,Y 127.861,Z 408.531,A -85,B 0,C 180,E1 -25821.478,E2 -25821.478} C_VEL
LIN {X 0,Y 130.723,Z 396.253,A -85,B 0,C 180,E1 -25823.833,E2 -25823.833} C_VEL
LIN {X 0,Y 133.11,Z 382.878,A -85,B 0,C 180,E1 -25825.671,E2 -25825.671} C_VEL
LIN {X 0,Y 134.795,Z 370.424,A -85,B 0,C 180,E1 -25826.823,E2 -25826.823} C_VEL
LIN {X 0,Y 138.576,Z 322.501,A -85,B 0,C 180,E1 -25829.55,E2 -25829.55} C_VEL
LIN {X 0,Y 133.137,Z 306.291,A -85,B 0,C 180,E1 -25832.189,E2 -25832.189} C_VEL
LIN {X 0,Y 125.913,Z 290.738,A -85,B 0,C 180,E1 -25835.657,E2 -25835.657} C_VEL
LIN {X 0,Y 117.234,Z 276.602,A -85,B 0,C 180,E1 -25840.046,E2 -25840.046} C_VEL
LIN {X 0,Y 115.625,Z 274.101,A -85,B 0,C 180,E1 -25840.984,E2 -25840.984} C_VEL
LIN {X 0,Y 115.254,Z 272.796,A -85,B 0,C 180,E1 -25841.873,E2 -25841.873} C_VEL
LIN {X 0,Y 114.946,Z 272.632,A -85,B 0,C 180,E1 -25847.807,E2 -25847.807} C_VEL
LIN {X 0,Y 114.9,Z 272.672,A -85,B 0,C 180,E1 -25853.504,E2 -25853.504} C_VEL
LIN {X 0,Y 114.823,Z 272.64,A -85,B 0,C 180,E1 -25861.081,E2 -25861.081} C_VEL
LIN {X 0,Y 114.813,Z 272.67,A -85,B 0,C 180,E1 -25867.75,E2 -25867.75} C_VEL
LIN {X 0,Y 114.837,Z 272.681,A -85,B 0,C 180,E1 -25872.782,E2 -25872.782} C_VEL
LIN {X 0,Y 114.863,Z 272.66,A -85,B 0,C 180,E1 -25877.732,E2 -25877.732} C_VEL
LIN {X 0,Y 114.873,Z 272.668,A -85,B 0,C 180,E1 -25882.697,E2 -25882.697} C_VEL
LIN {X 0,Y 114.847,Z 272.677,A -85,B 0,C 180,E1 -25888.96,E2 -25888.96} C_VEL
LIN {X 0,Y 114.913,Z 272.656,A -85,B 0,C 180,E1 -25896.56,E2 -25896.56} C_VEL
LIN {X 0,Y 114.963,Z 272.648,A -85,B 0,C 180,E1 -25902.227,E2 -25902.227} C_VEL
LIN {X 0,Y 115.306,Z 272.619,A -85,B 0,C 180,E1 -25909.488,E2 -25909.488} C_VEL
LIN {X 0,Y 115.496,Z 272.597,A -85,B 0,C 180,E1 -25916.535,E2 -25916.535} C_VEL
LIN {X 0,Y 115.981,Z 272.522,A -85,B 0,C 180,E1 -25920.023,E2 -25920.023} C_VEL
LIN {X 0,Y 115.359,Z 272.552,A -85,B 0,C 180,E1 -25927.021,E2 -25927.021} C_VEL
LIN {X 0,Y 115.224,Z 272.633,A -85,B 0,C 180,E1 -25932.578,E2 -25932.578} C_VEL
LIN {X 0,Y 114.989,Z 272.614,A -85,B 0,C 180,E1 -25937.817,E2 -25937.817} C_VEL
LIN {X 0,Y 114.952,Z 272.664,A -85,B 0,C 180,E1 -25943.485,E2 -25943.485} C_VEL
LIN {X 0,Y 114.885,Z 272.652,A -85,B 0,C 180,E1 -25951.07,E2 -25951.07} C_VEL
LIN {X 0,Y 114.841,Z 272.809,A -85,B 0,C 180,E1 -25953.708,E2 -25953.708} C_VEL
LIN {X 0,Y 115.132,Z 273.943,A -85,B 0,C 180,E1 -25954.536,E2 -25954.536} C_VEL
LIN {X 0,Y 117.019,Z 276.926,A -85,B 0,C 180,E1 -25955.669,E2 -25955.669} C_VEL
LIN {X 0,Y 123.872,Z 288.77,A -85,B 0,C 180,E1 -25959.293,E2 -25959.293} C_VEL
LIN {X 0,Y 128.997,Z 298.595,A -85,B 0,C 180,E1 -25961.76,E2 -25961.76} C_VEL
